C01824=1190.951,366.071,-77.906,-176.070,8.337,148.500
C01825=1190.946,366.351,-77.944,-176.068,8.340,148.500
C01826=1190.942,366.633,-77.983,-176.066,8.344,148.501
C01827=1190.937,366.914,-78.021,-176.065,8.348,148.501
C01828=1190.932,367.161,-78.055,-176.063,8.351,148.502
C01829=1190.929,367.409,-78.090,-176.062,8.354,148.502
C01830=1190.925,367.657,-78.123,-176.060,8.358,148.502
C01831=1190.920,367.904,-78.157,-176.058,8.361,148.503
C01832=1190.917,368.152,-78.191,-176.057,8.364,148.503
C01833=1190.913,368.400,-78.226,-176.055,8.368,148.504
C01834=1190.909,368.647,-78.260,-176.053,8.371,148.504
C01835=1190.904,368.895,-78.294,-176.052,8.374,148.504
C01836=1190.901,369.143,-78.328,-176.050,8.378,148.505
C01837=1190.896,369.390,-78.362,-176.049,8.381,148.505
C01838=1190.893,369.638,-78.396,-176.047,8.385,148.506
C01839=1190.888,369.885,-78.431,-176.046,8.387,148.506
C01840=1190.885,370.134,-78.464,-176.044,8.391,148.507
C01841=1190.880,370.381,-78.499,-176.043,8.394,148.507
C01842=1190.876,370.628,-78.533,-176.041,8.397,148.508
C01843=1190.872,370.876,-78.568,-176.040,8.401,148.508
C01844=1190.869,371.123,-78.602,-176.038,8.404,148.508
C01845=1190.864,371.371,-78.636,-176.037,8.408,148.509
C01846=1190.861,371.619,-78.670,-176.036,8.411,148.509
C01847=1190.856,371.866,-78.705,-176.034,8.414,148.510
C01848=1190.852,372.114,-78.740,-176.033,8.417,148.510
C01849=1190.848,372.362,-78.773,-176.031,8.421,148.511
C01850=1190.843,372.609,-78.807,-176.030,8.424,148.511
C01851=1190.840,372.857,-78.841,-176.029,8.427,148.512
C01852=1190.836,373.105,-78.876,-176.027,8.430,148.512
C01853=1190.832,373.352,-78.910,-176.026,8.433,148.513
C01854=1190.828,373.600,-78.945,-176.025,8.437,148.513
C01855=1190.823,373.847,-78.979,-176.023,8.440,148.513
C01856=1190.820,374.095,-79.013,-176.022,8.444,148.514
C01857=1190.816,374.342,-79.048,-176.021,8.446,148.514
C01858=1190.812,374.591,-79.083,-176.020,8.450,148.515
C01859=1190.808,374.838,-79.116,-176.018,8.453,148.516
C01860=1190.804,375.086,-79.151,-176.017,8.456,148.516
C01861=1190.800,375.333,-79.185,-176.016,8.460,148.517
C01862=1190.796,375.580,-79.220,-176.014,8.463,148.517
C01863=1190.792,375.828,-79.255,-176.013,8.466,148.518
C01864=1190.788,376.075,-79.289,-176.012,8.469,148.518
C01865=1190.784,376.323,-79.324,-176.011,8.473,148.519
C01866=1190.779,376.570,-79.358,-176.010,8.475,148.519
C01867=1190.776,376.818,-79.393,-176.009,8.478,148.520
C01868=1190.772,377.066,-79.427,-176.007,8.482,148.520
C01869=1190.768,377.314,-79.462,-176.006,8.485,148.521
C01870=1190.764,377.561,-79.496,-176.005,8.488,148.521
C01871=1190.760,377.808,-79.531,-176.004,8.492,148.522
C01872=1190.755,378.056,-79.566,-176.002,8.495,148.522
C01873=1190.752,378.304,-79.601,-176.002,8.498,148.523
C01874=1190.748,378.551,-79.634,-176.001,8.501,148.523
C01875=1190.744,378.799,-79.669,-175.999,8.505,148.524
C01876=1190.739,379.047,-79.704,-175.998,8.508,148.524
C01877=1190.735,379.294,-79.739,-175.997,8.510,148.525
C01878=1190.732,379.541,-79.773,-175.996,8.513,148.525
C01879=1190.728,379.789,-79.808,-175.995,8.517,148.526
C01880=1190.723,380.037,-79.842,-175.995,8.520,148.526
C01881=1190.719,380.284,-79.878,-175.993,8.523,148.527
C01882=1190.716,380.531,-79.912,-175.992,8.526,148.527
C01883=1190.712,380.779,-79.947,-175.991,8.530,148.528
C01884=1190.707,381.027,-79.981,-175.990,8.532,148.528
C01885=1190.703,381.274,-80.017,-175.989,8.535,148.529
C01886=1190.700,381.522,-80.051,-175.988,8.539,148.529
C01887=1190.696,381.770,-80.085,-175.988,8.542,148.530
C01888=1190.691,382.017,-80.120,-175.986,8.544,148.530
C01889=1190.687,382.265,-80.155,-175.986,8.548,148.531
C01890=1190.683,382.512,-80.190,-175.985,8.551,148.532
C01891=1190.680,382.760,-80.224,-175.984,8.554,148.532
C01892=1190.675,383.007,-80.259,-175.983,8.557,148.533
C01893=1190.671,383.255,-80.294,-175.982,8.560,148.533
C01894=1190.667,383.502,-80.329,-175.981,8.563,148.534
C01895=1190.663,383.750,-80.364,-175.980,8.566,148.534
C01896=1190.659,383.998,-80.399,-175.980,8.569,148.535
C01897=1190.656,384.244,-80.434,-175.979,8.572,148.535
C01898=1190.652,384.492,-80.468,-175.978,8.575,148.536
C01899=1190.647,384.740,-80.503,-175.977,8.578,148.537
C01900=1190.643,384.987,-80.538,-175.976,8.581,148.537
C01901=1190.639,385.235,-80.573,-175.976,8.584,148.538
C01902=1190.635,385.482,-80.608,-175.975,8.587,148.538
C01903=1190.631,385.730,-80.643,-175.974,8.591,148.539
C01904=1190.627,385.978,-80.678,-175.974,8.593,148.540
C01905=1190.624,386.225,-80.713,-175.973,8.596,148.540
C01906=1190.619,386.472,-80.747,-175.972,8.599,148.541
C01907=1190.615,386.720,-80.783,-175.971,8.602,148.541
C01908=1190.611,386.967,-80.817,-175.970,8.605,148.542
C01909=1190.607,387.215,-80.853,-175.970,8.608,148.542
C01910=1190.603,387.463,-80.888,-175.969,8.611,148.543
C01911=1190.599,387.710,-80.923,-175.969,8.614,148.544
C01912=1190.595,387.958,-80.958,-175.968,8.617,148.544
C01913=1190.591,388.205,-80.993,-175.968,8.619,148.545
C01914=1190.587,388.453,-81.028,-175.967,8.622,148.545
C01915=1190.584,388.700,-81.063,-175.966,8.625,148.546
C01916=1190.579,388.947,-81.097,-175.966,8.628,148.546
C01917=1190.576,389.195,-81.133,-175.965,8.631,148.547
C01918=1190.571,389.442,-81.167,-175.964,8.634,148.548
C01919=1190.567,389.690,-81.203,-175.964,8.636,148.548
C01920=1190.563,389.938,-81.237,-175.963,8.639,148.549
C01921=1190.559,390.185,-81.273,-175.962,8.642,148.549
C01922=1190.555,390.433,-81.307,-175.963,8.645,148.550
C01923=1190.552,390.680,-81.343,-175.962,8.648,148.551
C01924=1190.547,390.927,-81.378,-175.961,8.650,148.551
C01925=1190.543,391.175,-81.413,-175.961,8.653,148.552
C01926=1190.540,391.423,-81.449,-175.960,8.655,148.552
C01927=1190.535,391.670,-81.483,-175.960,8.659,148.553
C01928=1190.531,391.954,-81.524,-175.959,8.662,148.554
C01929=1190.527,392.237,-81.563,-175.958,8.665,148.554
C01930=1190.522,392.520,-81.604,-175.959,8.668,148.555
C01931=1190.517,392.804,-81.644,-175.958,8.671,148.555
C01932=1190.513,393.051,-81.679,-175.957,8.674,148.556
C01933=1190.510,393.299,-81.715,-175.957,8.676,148.557
C01934=1190.505,393.546,-81.749,-175.956,8.680,148.557
C01935=1190.501,393.794,-81.785,-175.956,8.682,148.558
C01936=1190.498,394.041,-81.820,-175.956,8.684,148.558
C01937=1190.493,394.289,-81.855,-175.955,8.687,148.559
C01938=1190.489,394.536,-81.890,-175.955,8.689,148.560
C01939=1190.486,394.784,-81.926,-175.954,8.693,148.560
C01940=1190.481,395.031,-81.960,-175.954,8.695,148.561
C01941=1190.478,395.279,-81.996,-175.954,8.697,148.561
C01942=1190.474,395.526,-82.031,-175.953,8.700,148.562
C01943=1190.469,395.774,-82.066,-175.953,8.703,148.562
C01944=1190.466,396.021,-82.102,-175.953,8.705,148.563
C01945=1190.462,396.269,-82.137,-175.952,8.708,148.564
C01946=1190.457,396.516,-82.173,-175.952,8.711,148.564
C01947=1190.453,396.764,-82.208,-175.952,8.713,148.565
C01948=1190.449,397.011,-82.243,-175.952,8.715,148.565
C01949=1190.445,397.258,-82.278,-175.951,8.718,148.566
C01950=1190.441,397.506,-82.313,-175.951,8.721,148.567
C01951=1190.438,397.754,-82.349,-175.951,8.723,148.567
C01952=1190.433,398.000,-82.384,-175.951,8.725,148.568
C01953=1190.430,398.248,-82.420,-175.950,8.728,148.568
C01954=1190.426,398.496,-82.454,-175.950,8.731,148.569
C01955=1190.421,398.743,-82.490,-175.950,8.733,148.570
C01956=1190.418,398.990,-82.525,-175.949,8.736,148.570
C01957=1190.414,399.238,-82.561,-175.949,8.738,148.571
C01958=1190.410,399.485,-82.596,-175.949,8.740,148.571
C01959=1190.405,399.733,-82.631,-175.949,8.744,148.572
C01960=1190.401,399.981,-82.667,-175.948,8.746,148.572
C01961=1190.398,400.228,-82.702,-175.948,8.748,148.573
C01962=1190.393,400.475,-82.737,-175.948,8.750,148.574
C01963=1190.390,400.722,-82.773,-175.948,8.753,148.574
C01964=1190.386,400.971,-82.808,-175.948,8.755,148.575
C01965=1190.382,401.218,-82.843,-175.948,8.757,148.575
C01966=1190.378,401.465,-82.879,-175.947,8.760,148.576
C01967=1190.374,401.712,-82.914,-175.947,8.763,148.576
C01968=1190.370,401.960,-82.950,-175.946,8.765,148.577
C01969=1190.365,402.208,-82.985,-175.947,8.768,148.578
C01970=1190.362,402.455,-83.020,-175.946,8.770,148.578
C01971=1190.358,402.703,-83.056,-175.946,8.772,148.579
C01972=1190.354,402.950,-83.091,-175.946,8.774,148.579
C01973=1190.350,403.197,-83.127,-175.946,8.777,148.580
C01974=1190.346,403.444,-83.162,-175.946,8.779,148.581
C01975=1190.342,403.692,-83.198,-175.945,8.781,148.581
C01976=1190.338,403.940,-83.233,-175.945,8.784,148.582
C01977=1190.334,404.187,-83.268,-175.945,8.786,148.582
C01978=1190.330,404.435,-83.304,-175.945,8.788,148.583
C01979=1190.326,404.682,-83.339,-175.944,8.791,148.583
C01980=1190.323,404.930,-83.375,-175.945,8.793,148.584
C01981=1190.318,405.177,-83.411,-175.944,8.795,148.584
C01982=1190.314,405.424,-83.446,-175.944,8.798,148.585
C01983=1190.310,405.672,-83.482,-175.944,8.800,148.585
C01984=1190.307,405.919,-83.517,-175.944,8.802,148.586
C01985=1190.302,406.166,-83.553,-175.944,8.804,148.586
C01986=1190.299,406.414,-83.587,-175.944,8.806,148.587
C01987=1190.294,406.662,-83.624,-175.944,8.808,148.588
C01988=1190.290,406.909,-83.659,-175.944,8.811,148.588
C01989=1190.286,407.156,-83.694,-175.943,8.813,148.589
C01990=1190.283,407.404,-83.730,-175.943,8.815,148.589
C01991=1190.279,407.651,-83.765,-175.943,8.818,148.590
C01992=1190.274,407.899,-83.801,-175.943,8.820,148.590
C01993=1190.270,408.146,-83.837,-175.943,8.822,148.591
C01994=1190.267,408.393,-83.872,-175.943,8.824,148.591
C01995=1190.263,408.641,-83.908,-175.943,8.826,148.592
C01996=1190.259,408.888,-83.943,-175.943,8.828,148.593
C01997=1190.254,409.135,-83.979,-175.942,8.831,148.593
C01998=1190.251,409.383,-84.015,-175.942,8.833,148.594
C01999=1190.247,409.630,-84.050,-175.942,8.835,148.594
C02000=1190.243,409.878,-84.086,-175.942,8.837,148.595
C02001=1190.240,410.125,-84.121,-175.942,8.839,148.595
C02002=1190.235,410.373,-84.157,-175.942,8.841,148.596
C02003=1190.231,410.620,-84.193,-175.942,8.844,148.596
C02004=1190.227,410.868,-84.228,-175.942,8.846,148.597
C02005=1190.224,411.115,-84.264,-175.941,8.848,148.597
C02006=1190.220,411.363,-84.299,-175.942,8.850,148.598
C02007=1190.215,411.610,-84.335,-175.941,8.852,148.598
C02008=1190.211,411.857,-84.371,-175.941,8.854,148.599
C02009=1190.208,412.105,-84.406,-175.941,8.856,148.599
C02010=1190.204,412.352,-84.442,-175.941,8.858,148.600
C02011=1190.199,412.599,-84.477,-175.941,8.860,148.600
C02012=1190.195,412.847,-84.513,-175.941,8.862,148.601
C02013=1190.192,413.094,-84.549,-175.941,8.865,148.601
C02014=1190.188,413.342,-84.584,-175.941,8.866,148.602
C02015=1190.184,413.590,-84.620,-175.941,8.868,148.602
C02016=1190.179,413.836,-84.655,-175.940,8.871,148.603
C02017=1190.176,414.084,-84.691,-175.940,8.873,148.603
C02018=1190.171,414.332,-84.727,-175.941,8.875,148.604
C02019=1190.168,414.579,-84.763,-175.941,8.877,148.605
C02020=1190.164,414.827,-84.798,-175.940,8.879,148.605
C02021=1190.160,415.074,-84.833,-175.941,8.881,148.606
C02022=1190.155,415.321,-84.870,-175.940,8.883,148.606
C02023=1190.152,415.569,-84.905,-175.940,8.885,148.607
C02024=1190.146,415.957,-84.961,-175.940,8.888,148.607
C02025=1190.142,416.344,-85.018,-175.940,8.891,148.608
C02026=1190.142,416.732,-85.072,-175.939,8.894,148.609
C02027=1190.144,417.119,-85.127,-175.939,8.897,148.610
C02028=1189.723,417.119,-85.168,-175.942,8.907,148.613
C02029=1189.720,416.730,-85.112,-175.943,8.905,148.613
C02030=1189.721,416.339,-85.057,-175.943,8.902,148.612
C02031=1189.724,415.948,-85.001,-175.943,8.898,148.611
C02032=1189.731,415.557,-84.945,-175.943,8.896,148.610
C02033=1189.734,415.310,-84.909,-175.943,8.893,148.610
C02034=1189.738,415.063,-84.872,-175.944,8.891,148.609
C02035=1189.743,414.816,-84.837,-175.943,8.890,148.609
C02036=1189.746,414.568,-84.801,-175.944,8.888,148.608
C02037=1189.750,414.321,-84.766,-175.944,8.885,148.608
C02038=1189.754,414.073,-84.730,-175.944,8.884,148.607
C02039=1189.758,413.825,-84.694,-175.944,8.882,148.607
C02040=1189.762,413.579,-84.659,-175.944,8.879,148.606
C02041=1189.766,413.331,-84.623,-175.944,8.877,148.606
C02042=1189.770,413.083,-84.587,-175.944,8.875,148.605
C02043=1189.774,412.836,-84.552,-175.944,8.873,148.605
C02044=1189.778,412.588,-84.516,-175.944,8.871,148.604
C02045=1189.782,412.342,-84.481,-175.944,8.869,148.604
C02046=1189.786,412.094,-84.445,-175.944,8.867,148.603
C02047=1189.790,411.846,-84.409,-175.944,8.865,148.603
C02048=1189.794,411.599,-84.374,-175.945,8.863,148.602
C02049=1189.797,411.351,-84.338,-175.945,8.860,148.602
C02050=1189.802,411.104,-84.302,-175.945,8.859,148.601
C02051=1189.806,410.857,-84.267,-175.945,8.857,148.601
C02052=1189.810,410.609,-84.231,-175.945,8.854,148.600
C02053=1189.813,410.362,-84.196,-175.945,8.852,148.599
C02054=1189.818,410.114,-84.160,-175.945,8.850,148.599
C02055=1189.822,409.867,-84.124,-175.945,8.848,148.598
C02056=1189.826,409.620,-84.089,-175.945,8.846,148.598
C02057=1189.829,409.372,-84.053,-175.945,8.844,148.597
C02058=1189.833,409.125,-84.018,-175.946,8.841,148.597
C02059=1189.838,408.877,-83.982,-175.946,8.839,148.596
C02060=1189.842,408.630,-83.947,-175.945,8.838,148.596
C02061=1189.845,408.382,-83.911,-175.946,8.835,148.595
C02062=1189.849,408.135,-83.875,-175.946,8.833,148.594
C02063=1189.853,407.887,-83.839,-175.946,8.830,148.594
C02064=1189.858,407.640,-83.804,-175.946,8.828,148.593
C02065=1189.861,407.393,-83.769,-175.946,8.826,148.593
C02066=1189.865,407.145,-83.733,-175.947,8.824,148.592
C02067=1189.869,406.898,-83.697,-175.946,8.822,148.592
C02068=1189.873,406.651,-83.662,-175.946,8.820,148.591
C02069=1189.877,406.403,-83.626,-175.946,8.817,148.591
C02070=1189.881,406.156,-83.591,-175.947,8.815,148.590
C02071=1189.885,405.908,-83.555,-175.947,8.813,148.590
C02072=1189.889,405.661,-83.520,-175.947,8.811,148.589
C02073=1189.892,405.414,-83.484,-175.947,8.808,148.589
C02074=1189.897,405.165,-83.449,-175.948,8.806,148.588
C02075=1189.901,404.918,-83.413,-175.947,8.803,148.587
C02076=1189.905,404.671,-83.378,-175.948,8.801,148.587
C02077=1189.909,404.424,-83.343,-175.948,8.799,148.586
C02078=1189.912,404.176,-83.307,-175.948,8.797,148.586
C02079=1189.916,403.929,-83.271,-175.948,8.794,148.585
C02080=1189.921,403.682,-83.236,-175.948,8.792,148.584
C02081=1189.925,403.434,-83.200,-175.948,8.790,148.584
C02082=1189.928,403.187,-83.165,-175.949,8.787,148.583
C02083=1189.932,402.938,-83.130,-175.949,8.785,148.583
C02084=1189.937,402.692,-83.095,-175.949,8.783,148.582
C02085=1189.940,402.444,-83.059,-175.949,8.780,148.582
C02086=1189.944,402.197,-83.024,-175.949,8.778,148.581
C02087=1189.948,401.949,-82.987,-175.949,8.776,148.581
C02088=1189.953,401.702,-82.952,-175.950,8.773,148.580
C02089=1189.956,401.455,-82.917,-175.950,8.771,148.580
C02090=1189.960,401.206,-82.882,-175.950,8.769,148.579
C02091=1189.965,400.960,-82.847,-175.950,8.766,148.578
C02092=1189.968,400.712,-82.811,-175.950,8.764,148.578
C02093=1189.972,400.465,-82.776,-175.950,8.762,148.577
C02094=1189.976,400.217,-82.740,-175.951,8.758,148.576
C02095=1189.981,399.969,-82.705,-175.951,8.756,148.576
C02096=1189.985,399.722,-82.669,-175.951,8.754,148.575
C02097=1189.988,399.474,-82.634,-175.952,8.752,148.575
C02098=1189.992,399.228,-82.599,-175.952,8.749,148.574
C02099=1189.996,398.980,-82.563,-175.952,8.747,148.574
C02100=1190.000,398.732,-82.528,-175.952,8.744,148.573
C02101=1190.004,398.484,-82.493,-175.953,8.741,148.573
C02102=1190.008,398.238,-82.458,-175.953,8.739,148.572
C02103=1190.012,397.990,-82.422,-175.953,8.737,148.571
C02104=1190.016,397.742,-82.387,-175.953,8.734,148.571
C02105=1190.021,397.495,-82.351,-175.954,8.731,148.570
C02106=1190.024,397.247,-82.316,-175.954,8.729,148.570
C02107=1190.028,397.000,-82.280,-175.954,8.727,148.569
C02108=1190.033,396.752,-82.246,-175.954,8.724,148.568
C02109=1190.036,396.505,-82.210,-175.955,8.721,148.568
C02110=1190.040,396.257,-82.175,-175.955,8.719,148.567
C02111=1190.044,396.011,-82.140,-175.955,8.716,148.567
C02112=1190.048,395.763,-82.105,-175.956,8.713,148.566
C02113=1190.052,395.515,-82.069,-175.956,8.711,148.565
C02114=1190.056,395.268,-82.034,-175.956,8.709,148.565
C02115=1190.060,395.020,-81.999,-175.957,8.705,148.564
C02116=1190.064,394.773,-81.964,-175.957,8.703,148.564
C02117=1190.068,394.526,-81.928,-175.957,8.701,148.563
C02118=1190.072,394.278,-81.893,-175.958,8.698,148.562
C02119=1190.076,394.030,-81.858,-175.958,8.695,148.562
C02120=1190.080,393.783,-81.823,-175.958,8.693,148.561
C02121=1190.083,393.536,-81.787,-175.959,8.690,148.561
C02122=1190.087,393.288,-81.752,-175.959,8.687,148.560
C02123=1190.092,393.041,-81.717,-175.960,8.684,148.560
C02124=1190.096,392.793,-81.682,-175.960,8.682,148.559
C02125=1190.100,392.510,-81.642,-175.961,8.679,148.558
C02126=1190.105,392.226,-81.601,-175.961,8.675,148.558
C02127=1190.109,391.942,-81.561,-175.962,8.672,148.557
C02128=1190.114,391.659,-81.520,-175.962,8.669,148.556
C02129=1190.118,391.411,-81.486,-175.963,8.667,148.556
C02130=1190.122,391.164,-81.450,-175.963,8.664,148.555
C02131=1190.126,390.916,-81.416,-175.964,8.661,148.555
C02132=1190.130,390.669,-81.380,-175.964,8.658,148.554
C02133=1190.134,390.421,-81.344,-175.964,8.656,148.553
C02134=1190.138,390.174,-81.311,-175.965,8.653,148.553
C02135=1190.141,389.927,-81.275,-175.966,8.649,148.552
C02136=1190.146,389.679,-81.241,-175.966,8.647,148.552
C02137=1190.150,389.432,-81.205,-175.967,8.644,148.551
C02138=1190.153,389.184,-81.170,-175.967,8.642,148.551
C02139=1190.158,388.937,-81.135,-175.968,8.639,148.550
C02140=1190.162,388.689,-81.100,-175.969,8.636,148.549
C02141=1190.165,388.441,-81.065,-175.969,8.633,148.549
C02142=1190.170,388.194,-81.030,-175.969,8.630,148.548
C02143=1190.174,387.946,-80.995,-175.970,8.627,148.547
C02144=1190.178,387.699,-80.960,-175.971,8.624,148.547
C02145=1190.182,387.452,-80.925,-175.971,8.622,148.546
C02146=1190.186,387.203,-80.890,-175.972,8.618,148.546
C02147=1190.190,386.957,-80.855,-175.973,8.615,148.545
C02148=1190.194,386.708,-80.820,-175.974,8.612,148.545
C02149=1190.198,386.462,-80.785,-175.974,8.610,148.544
C02150=1190.202,386.214,-80.750,-175.975,8.607,148.543
C02151=1190.205,385.966,-80.715,-175.975,8.604,148.543
C02152=1190.210,385.719,-80.680,-175.976,8.601,148.542
C02153=1190.213,385.471,-80.645,-175.977,8.598,148.542
C02154=1190.218,385.224,-80.610,-175.978,8.594,148.541
C02155=1190.222,384.977,-80.575,-175.978,8.592,148.541
C02156=1190.226,384.729,-80.540,-175.979,8.589,148.540
C02157=1190.229,384.481,-80.506,-175.980,8.586,148.540
C02158=1190.233,384.234,-80.471,-175.981,8.583,148.539
C02159=1190.238,383.986,-80.436,-175.982,8.580,148.538
C02160=1190.241,383.739,-80.401,-175.983,8.577,148.538
C02161=1190.246,383.491,-80.366,-175.983,8.574,148.537
C02162=1190.250,383.243,-80.331,-175.984,8.571,148.537
C02163=1190.253,382.997,-80.297,-175.985,8.568,148.536
C02164=1190.257,382.749,-80.262,-175.986,8.565,148.536
C02165=1190.262,382.501,-80.227,-175.987,8.562,148.535
C02166=1190.266,382.254,-80.192,-175.988,8.559,148.535
C02167=1190.270,382.006,-80.157,-175.989,8.556,148.534
C02168=1190.274,381.758,-80.122,-175.989,8.553,148.533
C02169=1190.277,381.511,-80.088,-175.990,8.549,148.533
C02170=1190.282,381.264,-80.053,-175.991,8.547,148.532
C02171=1190.286,381.016,-80.018,-175.993,8.543,148.532
C02172=1190.290,380.768,-79.984,-175.994,8.540,148.531
C02173=1190.294,380.521,-79.948,-175.994,8.536,148.531
C02174=1190.298,380.274,-79.914,-175.996,8.534,148.530
C02175=1190.302,380.025,-79.880,-175.996,8.531,148.530
C02176=1190.306,379.779,-79.844,-175.997,8.528,148.529
C02177=1190.310,379.530,-79.809,-175.998,8.525,148.529
C02178=1190.314,379.283,-79.776,-176.000,8.521,148.528
C02179=1190.318,379.035,-79.741,-176.001,8.518,148.527
C02180=1190.322,378.788,-79.706,-176.002,8.515,148.527
C02181=1190.326,378.540,-79.671,-176.003,8.512,148.526
C02182=1190.330,378.293,-79.637,-176.003,8.509,148.526
C02183=1190.334,378.045,-79.602,-176.005,8.505,148.525
C02184=1190.338,377.798,-79.568,-176.006,8.502,148.525
C02185=1190.342,377.550,-79.533,-176.007,8.499,148.524
C02186=1190.346,377.302,-79.499,-176.008,8.496,148.524
C02187=1190.350,377.055,-79.463,-176.009,8.492,148.523
C02188=1190.354,376.808,-79.429,-176.011,8.489,148.523
C02189=1190.358,376.560,-79.395,-176.011,8.486,148.522
C02190=1190.362,376.312,-79.360,-176.013,8.483,148.522
C02191=1190.367,376.065,-79.326,-176.014,8.480,148.521
C02192=1190.370,375.817,-79.291,-176.015,8.477,148.521
C02193=1190.374,375.570,-79.257,-176.017,8.473,148.520
C02194=1190.378,375.322,-79.222,-176.018,8.470,148.520
C02195=1190.382,375.074,-79.188,-176.019,8.467,148.519
C02196=1190.386,374.826,-79.153,-176.020,8.463,148.519
C02197=1190.391,374.579,-79.118,-176.022,8.460,148.518
C02198=1190.394,374.332,-79.084,-176.023,8.457,148.518
C02199=1190.398,374.084,-79.050,-176.024,8.454,148.517
C02200=1190.402,373.837,-79.016,-176.026,8.451,148.517
C02201=1190.406,373.589,-78.981,-176.027,8.447,148.516
C02202=1190.411,373.342,-78.946,-176.028,8.444,148.516
C02203=1190.414,373.094,-78.912,-176.030,8.441,148.516
C02204=1190.418,372.846,-78.878,-176.031,8.437,148.515
C02205=1190.422,372.599,-78.843,-176.033,8.434,148.515
C02206=1190.426,372.351,-78.809,-176.034,8.431,148.514
C02207=1190.431,372.103,-78.775,-176.036,8.427,148.514
C02208=1190.434,371.855,-78.741,-176.036,8.424,148.513
C02209=1190.439,371.608,-78.707,-176.038,8.421,148.513
C02210=1190.442,371.360,-78.672,-176.039,8.418,148.512
C02211=1190.447,371.113,-78.638,-176.041,8.414,148.512
C02212=1190.451,370.866,-78.604,-176.042,8.411,148.511
C02213=1190.455,370.617,-78.569,-176.044,8.408,148.511
C02214=1190.458,370.370,-78.535,-176.045,8.405,148.510
C02215=1190.463,370.123,-78.501,-176.047,8.401,148.510
C02216=1190.466,369.875,-78.467,-176.048,8.398,148.510
C02217=1190.471,369.627,-78.433,-176.050,8.395,148.509
C02218=1190.474,369.379,-78.399,-176.052,8.391,148.509
C02219=1190.479,369.132,-78.364,-176.052,8.388,148.508
C02220=1190.483,368.885,-78.330,-176.054,8.384,148.508
C02221=1190.487,368.637,-78.295,-176.055,8.382,148.507
C02222=1190.491,368.389,-78.262,-176.057,8.378,148.507
C02223=1190.495,368.141,-78.228,-176.059,8.374,148.506
C02224=1190.499,367.894,-78.194,-176.060,8.371,148.506
C02225=1190.503,367.646,-78.159,-176.062,8.368,148.506
C02226=1190.507,367.398,-78.126,-176.063,8.365,148.505
C02227=1190.511,367.150,-78.091,-176.065,8.361,148.505
C02228=1190.515,366.903,-78.057,-176.067,8.358,148.504
C02229=1190.520,366.623,-78.019,-176.069,8.354,148.504
C02230=1190.524,366.341,-77.980,-176.071,8.351,148.504
C02231=1190.530,366.060,-77.942,-176.072,8.347,148.503
C02232=1190.534,365.778,-77.903,-176.074,8.343,148.503
C02233=1190.538,365.531,-77.869,-176.076,8.340,148.502
C02234=1190.541,365.283,-77.835,-176.078,8.336,148.502
C02235=1190.546,365.035,-77.801,-176.079,8.333,148.501
C02236=1190.550,364.788,-77.767,-176.081,8.330,148.501
C02237=1190.554,364.541,-77.734,-176.083,8.326,148.501
C02238=1190.558,364.293,-77.699,-176.085,8.323,148.500
C02239=1190.562,364.045,-77.665,-176.086,8.320,148.500
C02240=1190.567,363.797,-77.631,-176.088,8.316,148.499
C02241=1190.570,363.550,-77.597,-176.090,8.313,148.499
C02242=1190.574,363.302,-77.564,-176.092,8.309,148.499
C02243=1190.578,363.055,-77.530,-176.093,8.306,148.498
C02244=1190.583,362.807,-77.496,-176.095,8.303,148.498
C02245=1190.586,362.559,-77.462,-176.097,8.299,148.498
C02246=1190.590,362.311,-77.429,-176.099,8.296,148.497
C02247=1190.595,362.064,-77.394,-176.100,8.293,148.497
C02248=1190.599,361.816,-77.361,-176.102,8.289,148.497
C02249=1190.602,361.568,-77.327,-176.104,8.286,148.496
C02250=1190.606,361.320,-77.294,-176.106,8.282,148.496
C02251=1190.611,361.073,-77.259,-176.107,8.280,148.495
C02252=1190.615,360.825,-77.226,-176.109,8.276,148.495
C02253=1190.619,360.578,-77.192,-176.111,8.273,148.495
C02254=1190.622,360.330,-77.159,-176.114,8.269,148.495
C02255=1190.627,360.082,-77.125,-176.115,8.266,148.494
C02256=1190.631,359.835,-77.091,-176.117,8.263,148.494
C02257=1190.635,359.587,-77.058,-176.119,8.260,148.494
C02258=1190.639,359.340,-77.024,-176.121,8.256,148.493
C02259=1190.643,359.091,-76.990,-176.123,8.253,148.493
C02260=1190.647,358.843,-76.957,-176.125,8.249,148.492
C02261=1190.651,358.596,-76.923,-176.127,8.246,148.492
C02262=1190.655,358.348,-76.890,-176.128,8.243,148.492
C02263=1190.659,358.101,-76.857,-176.130,8.240,148.492
C02264=1190.663,357.854,-76.823,-176.132,8.236,148.491
C02265=1190.667,357.605,-76.789,-176.134,8.233,148.491
C02266=1190.672,357.357,-76.756,-176.136,8.229,148.491
C02267=1190.676,357.109,-76.722,-176.138,8.226,148.490
C02268=1190.680,356.862,-76.689,-176.141,8.222,148.490
C02269=1190.684,356.615,-76.655,-176.142,8.219,148.490
C02270=1190.688,356.367,-76.622,-176.144,8.216,148.489
C02271=1190.692,356.119,-76.589,-176.146,8.213,148.489
C02272=1190.696,355.871,-76.554,-176.148,8.209,148.489
C02273=1190.700,355.623,-76.521,-176.150,8.206,148.489
C02274=1190.704,355.376,-76.488,-176.152,8.202,148.488
C02275=1190.708,355.128,-76.455,-176.154,8.199,148.488
C02276=1190.712,354.880,-76.422,-176.157,8.196,148.488
C02277=1190.717,354.632,-76.389,-176.158,8.193,148.487
C02278=1190.720,354.385,-76.355,-176.160,8.190,148.487
C02279=1190.725,354.138,-76.321,-176.162,8.186,148.487
C02280=1190.729,353.890,-76.288,-176.164,8.183,148.486
C02281=1190.732,353.641,-76.255,-176.166,8.179,148.486
C02282=1190.736,353.394,-76.222,-176.169,8.176,148.486
C02283=1190.741,353.146,-76.189,-176.171,8.173,148.486
C02284=1190.745,352.898,-76.155,-176.172,8.170,148.485
C02285=1190.749,352.650,-76.122,-176.174,8.167,148.485
C02286=1190.753,352.403,-76.089,-176.177,8.163,148.485
C02287=1190.757,352.155,-76.056,-176.179,8.160,148.485
C02288=1190.761,351.907,-76.023,-176.181,8.156,148.484
C02289=1190.765,351.660,-75.990,-176.183,8.153,148.484
C02290=1190.769,351.412,-75.956,-176.185,8.150,148.484
C02291=1190.774,351.164,-75.923,-176.187,8.146,148.484
C02292=1190.778,350.916,-75.890,-176.189,8.144,148.483
C02293=1190.782,350.669,-75.857,-176.191,8.140,148.483
C02294=1190.786,350.421,-75.824,-176.193,8.137,148.483
C02295=1190.790,350.173,-75.791,-176.195,8.133,148.483
C02296=1190.794,349.925,-75.757,-176.198,8.130,148.482
C02297=1190.798,349.678,-75.724,-176.200,8.127,148.482
C02298=1190.803,349.429,-75.692,-176.202,8.123,148.482
C02299=1190.807,349.182,-75.659,-176.204,8.121,148.482
C02300=1190.811,348.934,-75.626,-176.206,8.117,148.481
C02301=1190.815,348.686,-75.593,-176.208,8.114,148.481
C02302=1190.819,348.439,-75.560,-176.210,8.111,148.481
C02303=1190.823,348.191,-75.527,-176.212,8.107,148.481
C02304=1190.827,347.943,-75.494,-176.215,8.104,148.480
C02305=1190.831,347.695,-75.461,-176.217,8.101,148.480
C02306=1190.836,347.447,-75.428,-176.219,8.098,148.480
C02307=1190.840,347.199,-75.395,-176.221,8.095,148.480
C02308=1190.843,346.952,-75.362,-176.223,8.092,148.480
C02309=1190.848,346.704,-75.330,-176.225,8.088,148.479
C02310=1190.852,346.456,-75.297,-176.228,8.085,148.479
C02311=1190.856,346.208,-75.263,-176.230,8.082,148.479
C02312=1190.860,345.960,-75.231,-176.232,8.078,148.479
C02313=1190.864,345.712,-75.198,-176.234,8.075,148.478
C02314=1190.868,345.465,-75.165,-176.236,8.072,148.478
C02315=1190.873,345.218,-75.133,-176.238,8.069,148.478
C02316=1190.877,344.969,-75.100,-176.240,8.066,148.478
C02317=1190.881,344.722,-75.067,-176.243,8.063,148.478
C02318=1190.885,344.474,-75.035,-176.245,8.059,148.477
C02319=1190.889,344.226,-75.002,-176.247,8.056,148.477
C02320=1190.893,343.978,-74.969,-176.249,8.053,148.477
C02321=1190.898,343.730,-74.936,-176.251,8.050,148.477
C02322=1190.901,343.482,-74.904,-176.253,8.047,148.477
C02323=1190.905,343.234,-74.871,-176.256,8.043,148.476
C02324=1190.910,342.986,-74.838,-176.258,8.040,148.476
C02325=1190.915,342.739,-74.806,-176.260,8.037,148.476
C02326=1190.918,342.491,-74.774,-176.262,8.033,148.476
C02327=1190.922,342.244,-74.740,-176.265,8.030,148.475
C02328=1190.927,341.995,-74.708,-176.267,8.028,148.476
C02329=1190.930,341.748,-74.675,-176.269,8.025,148.475
C02330=1190.934,341.499,-74.643,-176.271,8.021,148.475
C02331=1190.939,341.252,-74.611,-176.273,8.018,148.475
C02332=1190.943,341.004,-74.578,-176.276,8.015,148.475
C02333=1190.947,340.726,-74.542,-176.278,8.011,148.474
C02334=1190.953,340.447,-74.505,-176.281,8.007,148.474
C02335=1190.957,340.168,-74.469,-176.283,8.004,148.474
C02336=1190.962,339.889,-74.432,-176.286,8.001,148.474
C02337=1190.965,339.642,-74.400,-176.288,7.997,148.474
C02338=1190.970,339.393,-74.367,-176.290,7.994,148.474
C02339=1190.974,339.145,-74.335,-176.292,7.991,148.473
C02340=1190.978,338.898,-74.303,-176.295,7.987,148.473
C02341=1190.982,338.650,-74.270,-176.297,7.985,148.473
C02342=1190.986,338.402,-74.238,-176.299,7.982,148.473
C02343=1190.990,338.154,-74.205,-176.301,7.979,148.473
C02344=1190.995,337.907,-74.174,-176.303,7.975,148.472
C02345=1190.999,337.659,-74.141,-176.306,7.972,148.472
C02346=1191.003,337.410,-74.109,-176.308,7.969,148.472
C02347=1191.007,337.163,-74.076,-176.311,7.966,148.472
C02348=1191.011,336.914,-74.044,-176.312,7.963,148.472
C02349=1191.016,336.667,-74.012,-176.315,7.960,148.472
C02350=1191.020,336.419,-73.980,-176.317,7.957,148.472
C02351=1191.024,336.171,-73.947,-176.320,7.953,148.471
C02352=1191.027,335.923,-73.915,-176.322,7.950,148.471
C02353=1191.032,335.676,-73.883,-176.324,7.947,148.471
C02354=1191.036,335.428,-73.851,-176.327,7.944,148.471
C02355=1191.040,335.179,-73.819,-176.328,7.941,148.471
C02356=1191.044,334.931,-73.787,-176.331,7.938,148.471
C02357=1191.049,334.684,-73.754,-176.333,7.935,148.471
C02358=1191.053,334.436,-73.723,-176.336,7.932,148.470
C02359=1191.057,334.188,-73.690,-176.338,7.928,148.470
C02360=1191.061,333.940,-73.659,-176.340,7.925,148.470
C02361=1191.065,333.692,-73.627,-176.342,7.923,148.470
C02362=1191.069,333.444,-73.594,-176.344,7.919,148.470
C02363=1191.073,333.196,-73.563,-176.347,7.916,148.470
C02364=1191.078,332.948,-73.530,-176.349,7.913,148.470
C02365=1191.082,332.700,-73.499,-176.352,7.910,148.469
C02366=1191.086,332.452,-73.467,-176.354,7.907,148.469
C02367=1191.091,332.205,-73.435,-176.357,7.903,148.469
C02368=1191.094,331.957,-73.403,-176.359,7.901,148.469
C02369=1191.098,331.709,-73.371,-176.361,7.898,148.469
C02370=1191.103,331.461,-73.339,-176.363,7.895,148.469
C02371=1191.107,331.213,-73.307,-176.366,7.892,148.469
C02372=1191.111,330.965,-73.275,-176.368,7.888,148.469
C02373=1191.116,330.717,-73.243,-176.371,7.885,148.469
C02374=1191.119,330.469,-73.211,-176.372,7.883,148.468
C02375=1191.124,330.222,-73.180,-176.375,7.879,148.468
C02376=1191.128,329.973,-73.147,-176.377,7.876,148.468
C02377=1191.132,329.725,-73.116,-176.380,7.873,148.468
C02378=1191.136,329.478,-73.084,-176.382,7.870,148.468
C02379=1191.140,329.229,-73.053,-176.385,7.867,148.468
C02380=1191.145,328.981,-73.020,-176.386,7.864,148.468
C02381=1191.149,328.734,-72.989,-176.389,7.861,148.468
C02382=1191.153,328.486,-72.957,-176.391,7.858,148.467
C02383=1191.157,328.238,-72.926,-176.394,7.855,148.467
C02384=1191.162,327.989,-72.894,-176.396,7.852,148.467
C02385=1191.165,327.741,-72.862,-176.399,7.849,148.467
C02386=1191.170,327.494,-72.831,-176.401,7.846,148.467
C02387=1191.173,327.246,-72.799,-176.403,7.843,148.467
C02388=1191.178,326.998,-72.768,-176.406,7.840,148.467
C02389=1191.182,326.750,-72.736,-176.408,7.837,148.467
C02390=1191.187,326.502,-72.704,-176.410,7.833,148.467
C02391=1191.190,326.254,-72.672,-176.413,7.830,148.467
C02392=1191.194,326.006,-72.641,-176.415,7.828,148.466
C02393=1191.199,325.758,-72.610,-176.418,7.825,148.466
C02394=1191.202,325.510,-72.578,-176.420,7.822,148.466
C02395=1191.207,325.262,-72.547,-176.422,7.819,148.466
C02396=1191.211,325.014,-72.515,-176.425,7.815,148.466
C02397=1191.216,324.767,-72.483,-176.427,7.812,148.466
C02398=1191.220,324.518,-72.452,-176.429,7.810,148.466
C02399=1191.224,324.271,-72.421,-176.432,7.807,148.466
C02400=1191.228,324.022,-72.389,-176.434,7.803,148.466
C02401=1191.232,323.775,-72.358,-176.437,7.800,148.466
C02402=1191.236,323.527,-72.326,-176.439,7.797,148.465
C02403=1191.241,323.279,-72.295,-176.442,7.794,148.465
C02404=1191.244,323.031,-72.263,-176.444,7.792,148.466
C02405=1191.249,322.783,-72.233,-176.446,7.789,148.465
C02406=1191.253,322.535,-72.201,-176.449,7.786,148.465
C02407=1191.257,322.287,-72.170,-176.451,7.782,148.465
C02408=1191.261,322.039,-72.138,-176.454,7.779,148.465
C02409=1191.266,321.791,-72.107,-176.455,7.777,148.465
C02410=1191.269,321.543,-72.076,-176.458,7.774,148.465
C02411=1191.274,321.295,-72.045,-176.461,7.771,148.465
C02412=1191.278,321.047,-72.013,-176.463,7.767,148.465
C02413=1191.282,320.799,-71.982,-176.466,7.764,148.465
C02414=1191.286,320.550,-71.951,-176.468,7.761,148.465
C02415=1191.291,320.303,-71.920,-176.470,7.759,148.465
C02416=1191.295,320.054,-71.888,-176.473,7.756,148.465
C02417=1191.299,319.807,-71.857,-176.475,7.752,148.464
C02418=1191.304,319.559,-71.826,-176.478,7.749,148.464
C02419=1191.308,319.310,-71.795,-176.480,7.746,148.464
C02420=1191.312,319.063,-71.764,-176.482,7.744,148.464
C02421=1191.316,318.814,-71.733,-176.485,7.741,148.464
C02422=1191.321,318.566,-71.702,-176.487,7.738,148.464
C02423=1191.325,318.317,-71.671,-176.490,7.735,148.464
C02424=1191.329,318.070,-71.639,-176.493,7.732,148.464
C02425=1191.333,317.822,-71.609,-176.495,7.728,148.464
C02426=1191.337,317.574,-71.578,-176.497,7.726,148.464
C02427=1191.341,317.326,-71.546,-176.500,7.723,148.464
C02428=1191.346,317.078,-71.516,-176.502,7.720,148.464
C02429=1191.350,316.830,-71.484,-176.505,7.717,148.464
C02430=1191.354,316.582,-71.454,-176.507,7.714,148.464
C02431=1191.358,316.333,-71.423,-176.509,7.711,148.464
C02432=1191.362,316.086,-71.392,-176.512,7.708,148.464
C02433=1191.366,315.838,-71.361,-176.514,7.705,148.464
C02434=1191.370,315.590,-71.330,-176.517,7.702,148.463
C02435=1191.375,315.342,-71.299,-176.519,7.699,148.463
C02436=1191.380,315.094,-71.268,-176.521,7.697,148.463
C02437=1191.384,314.817,-71.234,-176.525,7.693,148.463
C02438=1191.389,314.541,-71.200,-176.527,7.690,148.463
C02439=1191.393,314.264,-71.165,-176.530,7.687,148.463
C02440=1191.398,313.988,-71.131,-176.532,7.684,148.463
C02441=1191.402,313.740,-71.100,-176.535,7.681,148.463
C02442=1191.407,313.492,-71.069,-176.537,7.677,148.463
C02443=1191.411,313.244,-71.038,-176.540,7.674,148.463
C02444=1191.414,312.995,-71.008,-176.542,7.672,148.463
C02445=1191.419,312.748,-70.977,-176.545,7.669,148.463
C02446=1191.424,312.500,-70.946,-176.547,7.666,148.463
C02447=1191.428,312.251,-70.915,-176.550,7.663,148.463
C02448=1191.432,312.003,-70.885,-176.552,7.660,148.463
C02449=1191.436,311.755,-70.854,-176.555,7.657,148.463
C02450=1191.441,311.507,-70.824,-176.557,7.654,148.463
C02451=1191.444,311.259,-70.793,-176.560,7.651,148.463
C02452=1191.449,311.011,-70.762,-176.562,7.648,148.463
C02453=1191.453,310.763,-70.732,-176.565,7.645,148.463
C02454=1191.457,310.515,-70.702,-176.567,7.643,148.463
C02455=1191.461,310.266,-70.671,-176.569,7.640,148.463
C02456=1191.466,310.018,-70.640,-176.572,7.637,148.463
C02457=1191.470,309.771,-70.610,-176.575,7.634,148.463
C02458=1191.475,309.523,-70.579,-176.576,7.631,148.463
C02459=1191.478,309.274,-70.549,-176.579,7.628,148.463
C02460=1191.482,309.026,-70.518,-176.582,7.625,148.463
C02461=1191.487,308.778,-70.488,-176.585,7.622,148.463
C02462=1191.491,308.530,-70.458,-176.587,7.619,148.463
C02463=1191.496,308.282,-70.427,-176.589,7.617,148.462
C02464=1191.499,308.034,-70.396,-176.592,7.614,148.462
C02465=1191.504,307.785,-70.366,-176.594,7.611,148.462
C02466=1191.508,307.538,-70.336,-176.597,7.608,148.462
C02467=1191.513,307.290,-70.305,-176.599,7.605,148.463
C02468=1191.517,307.042,-70.275,-176.602,7.602,148.463
C02469=1191.521,306.793,-70.245,-176.604,7.599,148.462
C02470=1191.525,306.545,-70.214,-176.607,7.596,148.462
C02471=1191.529,306.297,-70.184,-176.609,7.594,148.462
C02472=1191.534,306.048,-70.154,-176.612,7.591,148.462
C02473=1191.538,305.801,-70.124,-176.614,7.588,148.462
C02474=1191.543,305.553,-70.093,-176.617,7.585,148.462
C02475=1191.547,305.305,-70.064,-176.619,7.582,148.462
C02476=1191.551,305.057,-70.033,-176.622,7.579,148.462
C02477=1191.555,304.808,-70.003,-176.624,7.576,148.462
C02478=1191.560,304.560,-69.972,-176.627,7.573,148.462
C02479=1191.564,304.312,-69.942,-176.630,7.570,148.462
C02480=1191.568,304.064,-69.913,-176.632,7.568,148.462
C02481=1191.572,303.816,-69.882,-176.634,7.565,148.462
C02482=1191.576,303.568,-69.852,-176.637,7.562,148.462
C02483=1191.581,303.320,-69.822,-176.639,7.559,148.462
C02484=1191.585,303.071,-69.792,-176.642,7.557,148.462
C02485=1191.590,302.823,-69.761,-176.644,7.554,148.462
C02486=1191.593,302.574,-69.732,-176.647,7.551,148.462
C02487=1191.597,302.327,-69.701,-176.650,7.548,148.462
C02488=1191.602,302.078,-69.671,-176.652,7.545,148.462
C02489=1191.606,301.831,-69.641,-176.654,7.542,148.462
C02490=1191.610,301.582,-69.612,-176.657,7.539,148.462
C02491=1191.615,301.334,-69.582,-176.660,7.536,148.462
C02492=1191.619,301.086,-69.551,-176.662,7.534,148.462
C02493=1191.623,300.838,-69.522,-176.664,7.531,148.462
C02494=1191.628,300.590,-69.491,-176.667,7.528,148.462
C02495=1191.632,300.342,-69.462,-176.669,7.526,148.462
C02496=1191.636,300.093,-69.432,-176.672,7.523,148.463
C02497=1191.641,299.845,-69.402,-176.675,7.520,148.463
C02498=1191.645,299.597,-69.372,-176.677,7.517,148.463
C02499=1191.649,299.349,-69.343,-176.679,7.514,148.463
C02500=1191.654,299.101,-69.312,-176.682,7.511,148.462
C02501=1191.658,298.853,-69.282,-176.684,7.508,148.462
C02502=1191.662,298.604,-69.253,-176.687,7.505,148.462
C02503=1191.666,298.356,-69.224,-176.689,7.503,148.463
C02504=1191.671,298.108,-69.193,-176.692,7.500,148.463
C02505=1191.675,297.860,-69.163,-176.695,7.497,148.463
C02506=1191.679,297.612,-69.134,-176.697,7.494,148.463
C02507=1191.684,297.363,-69.104,-176.700,7.492,148.463
C02508=1191.687,297.116,-69.074,-176.702,7.489,148.463
C02509=1191.692,296.867,-69.044,-176.705,7.486,148.463
C02510=1191.697,296.619,-69.015,-176.707,7.484,148.463
C02511=1191.701,296.371,-68.985,-176.710,7.481,148.463
C02512=1191.705,296.122,-68.956,-176.713,7.478,148.463
C02513=1191.709,295.874,-68.926,-176.715,7.475,148.463
C02514=1191.713,295.626,-68.896,-176.717,7.472,148.463
C02515=1191.718,295.378,-68.866,-176.720,7.469,148.463
C02516=1191.722,295.130,-68.837,-176.723,7.466,148.463
C02517=1191.726,294.881,-68.807,-176.725,7.464,148.463
C02518=1191.730,294.633,-68.778,-176.728,7.461,148.463
C02519=1191.735,294.385,-68.748,-176.730,7.458,148.463
C02520=1191.739,294.136,-68.719,-176.733,7.455,148.463
C02521=1191.743,293.888,-68.689,-176.735,7.453,148.463
C02522=1191.747,293.640,-68.660,-176.737,7.450,148.463
C02523=1191.752,293.392,-68.631,-176.740,7.447,148.463
C02524=1191.757,293.144,-68.601,-176.742,7.445,148.463
C02525=1191.761,292.895,-68.571,-176.745,7.441,148.463
C02526=1191.765,292.647,-68.542,-176.748,7.438,148.463
C02527=1191.769,292.399,-68.512,-176.750,7.436,148.463
C02528=1191.774,292.151,-68.483,-176.753,7.433,148.463
C02529=1191.778,291.902,-68.454,-176.755,7.430,148.463
C02530=1191.782,291.654,-68.424,-176.758,7.427,148.463
C02531=1191.786,291.406,-68.395,-176.760,7.425,148.463
C02532=1191.791,291.158,-68.366,-176.763,7.422,148.463
C02533=1191.795,290.910,-68.336,-176.766,7.419,148.463
C02534=1191.799,290.662,-68.307,-176.768,7.417,148.463
C02535=1191.804,290.413,-68.278,-176.770,7.414,148.463
C02536=1191.808,290.165,-68.249,-176.774,7.411,148.464
C02537=1191.812,289.916,-68.219,-176.776,7.409,148.464
C02538=1191.816,289.668,-68.190,-176.778,7.406,148.464
C02539=1191.821,289.421,-68.161,-176.781,7.403,148.464
C02540=1191.826,289.172,-68.132,-176.783,7.401,148.464
C02541=1191.829,288.897,-68.099,-176.786,7.398,148.464
C02542=1191.834,288.623,-68.067,-176.789,7.394,148.464
C02543=1191.840,288.349,-68.034,-176.792,7.391,148.464
C02544=1191.844,288.074,-68.002,-176.795,7.388,148.464
C02545=1191.849,287.826,-67.973,-176.797,7.386,148.464
C02546=1191.853,287.577,-67.945,-176.800,7.383,148.464
C02547=1191.857,287.329,-67.915,-176.802,7.380,148.464
C02548=1191.861,287.081,-67.886,-176.804,7.378,148.464
C02549=1191.866,286.832,-67.857,-176.808,7.375,148.464
C02550=1191.870,286.585,-67.828,-176.810,7.372,148.464
C02551=1191.874,286.336,-67.799,-176.813,7.370,148.465
C02552=1191.879,286.087,-67.770,-176.815,7.367,148.465
C02553=1191.883,285.839,-67.741,-176.818,7.364,148.465
C02554=1191.888,285.592,-67.712,-176.820,7.362,148.465
C02555=1191.892,285.343,-67.683,-176.823,7.359,148.465
C02556=1191.895,285.095,-67.654,-176.826,7.356,148.465
C02557=1191.900,284.846,-67.625,-176.828,7.353,148.465
C02558=1191.905,284.598,-67.596,-176.830,7.350,148.465
C02559=1191.909,284.350,-67.567,-176.833,7.347,148.465
C02560=1191.913,284.101,-67.538,-176.835,7.345,148.465
C02561=1191.917,283.854,-67.510,-176.838,7.342,148.465
C02562=1191.922,283.605,-67.481,-176.841,7.340,148.465
C02563=1191.926,283.357,-67.451,-176.843,7.337,148.465
C02564=1191.931,283.108,-67.423,-176.846,7.334,148.465
C02565=1191.935,282.861,-67.394,-176.848,7.332,148.465
C02566=1191.939,282.612,-67.365,-176.851,7.329,148.465
C02567=1191.943,282.363,-67.336,-176.854,7.326,148.465
C02568=1191.948,282.115,-67.308,-176.856,7.324,148.466
C02569=1191.952,281.867,-67.280,-176.858,7.321,148.466
C02570=1191.956,281.618,-67.250,-176.861,7.318,148.466
C02571=1191.961,281.370,-67.222,-176.863,7.316,148.466
C02572=1191.965,281.122,-67.193,-176.866,7.313,148.466
C02573=1191.969,280.873,-67.164,-176.869,7.310,148.466
C02574=1191.974,280.625,-67.136,-176.871,7.308,148.466
C02575=1191.978,280.377,-67.107,-176.874,7.305,148.466
C02576=1191.982,280.128,-67.078,-176.876,7.303,148.466
C02577=1191.987,279.880,-67.050,-176.879,7.300,148.466
C02578=1191.991,279.632,-67.021,-176.882,7.297,148.466
C02579=1191.995,279.383,-66.992,-176.884,7.295,148.466
C02580=1192.000,279.135,-66.964,-176.887,7.292,148.467
C02581=1192.004,278.887,-66.935,-176.889,7.290,148.467
C02582=1192.009,278.639,-66.907,-176.892,7.287,148.467
C02583=1192.013,278.390,-66.878,-176.895,7.284,148.467
C02584=1192.017,278.142,-66.850,-176.897,7.282,148.467
C02585=1192.021,277.894,-66.821,-176.899,7.279,148.467
C02586=1192.026,277.645,-66.792,-176.902,7.276,148.467
C02587=1192.031,277.397,-66.764,-176.905,7.274,148.467
C02588=1192.035,277.149,-66.736,-176.907,7.271,148.467
C02589=1192.039,276.900,-66.707,-176.910,7.269,148.467
C02590=1192.043,276.652,-66.679,-176.912,7.266,148.467
C02591=1192.048,276.404,-66.650,-176.915,7.263,148.467
C02592=1192.052,276.156,-66.622,-176.917,7.261,148.467
C02593=1192.056,275.907,-66.593,-176.920,7.258,148.468
C02594=1192.061,275.659,-66.566,-176.923,7.256,148.468
C02595=1192.065,275.410,-66.537,-176.925,7.253,148.468
C02596=1192.069,275.161,-66.509,-176.928,7.250,148.468
C02597=1192.074,274.913,-66.480,-176.930,7.247,148.468
C02598=1192.078,274.665,-66.452,-176.933,7.244,148.468
C02599=1192.083,274.417,-66.423,-176.935,7.243,148.468
C02600=1192.086,274.169,-66.395,-176.938,7.240,148.468
C02601=1192.091,273.921,-66.367,-176.940,7.237,148.468
C02602=1192.095,273.672,-66.339,-176.943,7.234,148.468
C02603=1192.100,273.424,-66.311,-176.946,7.231,148.468
C02604=1192.104,273.175,-66.282,-176.948,7.230,148.469
C02605=1192.108,272.927,-66.254,-176.951,7.227,148.469
C02606=1192.113,272.678,-66.226,-176.953,7.224,148.469
C02607=1192.117,272.430,-66.198,-176.956,7.221,148.469
C02608=1192.121,272.181,-66.170,-176.959,7.218,148.469
C02609=1192.126,271.933,-66.142,-176.961,7.217,148.469
C02610=1192.130,271.684,-66.114,-176.964,7.214,148.469
C02611=1192.135,271.437,-66.086,-176.966,7.211,148.469
C02612=1192.139,271.188,-66.057,-176.969,7.208,148.469
C02613=1192.143,270.940,-66.029,-176.971,7.207,148.470
C02614=1192.148,270.691,-66.001,-176.974,7.204,148.470
C02615=1192.152,270.443,-65.973,-176.977,7.201,148.470
C02616=1192.157,270.195,-65.945,-176.979,7.198,148.470
C02617=1192.161,269.946,-65.917,-176.982,7.195,148.470
C02618=1192.166,269.698,-65.889,-176.984,7.194,148.470
C02619=1192.169,269.449,-65.861,-176.987,7.191,148.470
C02620=1192.174,269.201,-65.833,-176.989,7.188,148.470
C02621=1192.178,268.952,-65.805,-176.992,7.185,148.470
C02622=1192.183,268.704,-65.778,-176.995,7.184,148.471
C02623=1192.187,268.456,-65.750,-176.997,7.181,148.471
C02624=1192.192,268.207,-65.721,-177.000,7.178,148.471
C02625=1192.196,267.959,-65.693,-177.002,7.175,148.471
C02626=1192.200,267.710,-65.666,-177.005,7.173,148.471
C02627=1192.205,267.462,-65.638,-177.008,7.171,148.471
C02628=1192.210,267.214,-65.610,-177.010,7.168,148.471
C02629=1192.214,266.965,-65.582,-177.012,7.165,148.471
C02630=1192.218,266.717,-65.555,-177.016,7.163,148.472
C02631=1192.222,266.468,-65.526,-177.018,7.161,148.472
C02632=1192.226,266.220,-65.499,-177.020,7.158,148.472
C02633=1192.232,265.972,-65.471,-177.023,7.155,148.472
C02634=1192.235,265.723,-65.443,-177.026,7.153,148.472
C02635=1192.240,265.475,-65.416,-177.028,7.151,148.472
C02636=1192.244,265.227,-65.388,-177.031,7.148,148.472
C02637=1192.248,264.978,-65.361,-177.033,7.145,148.472
C02638=1192.253,264.730,-65.333,-177.036,7.143,148.473
C02639=1192.258,264.482,-65.304,-177.038,7.141,148.473
C02640=1192.262,264.232,-65.277,-177.041,7.138,148.473
C02641=1192.266,263.984,-65.249,-177.044,7.135,148.473
C02642=1192.271,263.736,-65.222,-177.046,7.133,148.473
C02643=1192.275,263.487,-65.194,-177.049,7.130,148.473
C02644=1192.279,263.239,-65.167,-177.051,7.128,148.473
C02645=1192.285,262.966,-65.137,-177.054,7.125,148.473
C02646=1192.289,262.693,-65.106,-177.057,7.122,148.473
C02647=1192.294,262.421,-65.076,-177.060,7.119,148.474
C02648=1192.298,262.147,-65.046,-177.062,7.117,148.474
C02649=1192.303,261.899,-65.019,-177.065,7.114,148.474
C02650=1192.307,261.651,-64.991,-177.068,7.112,148.474
C02651=1192.312,261.402,-64.964,-177.070,7.109,148.474
C02652=1192.316,261.154,-64.936,-177.073,7.107,148.474
C02653=1192.320,260.905,-64.909,-177.076,7.104,148.475
C02654=1192.325,260.657,-64.881,-177.078,7.102,148.475
C02655=1192.329,260.409,-64.854,-177.081,7.099,148.475
C02656=1192.334,260.160,-64.826,-177.083,7.097,148.475
C02657=1192.338,259.912,-64.798,-177.086,7.094,148.475
C02658=1192.343,259.663,-64.771,-177.088,7.092,148.475
C02659=1192.347,259.415,-64.744,-177.091,7.090,148.475
C02660=1192.351,259.166,-64.717,-177.094,7.087,148.475
C02661=1192.356,258.918,-64.689,-177.096,7.084,148.476
C02662=1192.360,258.669,-64.662,-177.099,7.083,148.476
C02663=1192.365,258.421,-64.635,-177.102,7.080,148.476
C02664=1192.369,258.172,-64.607,-177.104,7.077,148.476
C02665=1192.373,257.924,-64.580,-177.107,7.075,148.476
C02666=1192.378,257.675,-64.553,-177.109,7.073,148.476
C02667=1192.383,257.427,-64.526,-177.112,7.070,148.476
C02668=1192.387,257.178,-64.499,-177.114,7.068,148.477
C02669=1192.391,256.930,-64.470,-177.117,7.065,148.477
C02670=1192.395,256.682,-64.444,-177.119,7.063,148.477
C02671=1192.400,256.433,-64.417,-177.123,7.060,148.477
C02672=1192.404,256.185,-64.390,-177.125,7.058,148.477
C02673=1192.409,255.936,-64.363,-177.127,7.056,148.477
C02674=1192.414,255.688,-64.336,-177.130,7.053,148.478
C02675=1192.418,255.438,-64.308,-177.132,7.051,148.478
C02676=1192.422,255.190,-64.281,-177.135,7.048,148.478
C02677=1192.426,254.942,-64.254,-177.138,7.046,148.478
C02678=1192.431,254.694,-64.227,-177.140,7.043,148.478
C02679=1192.435,254.445,-64.200,-177.143,7.041,148.478
C02680=1192.440,254.197,-64.173,-177.146,7.038,148.478
C02681=1192.445,253.948,-64.146,-177.148,7.036,148.479
C02682=1192.449,253.699,-64.118,-177.151,7.033,148.479
C02683=1192.453,253.451,-64.092,-177.153,7.031,148.479
C02684=1192.457,253.202,-64.065,-177.156,7.029,148.479
C02685=1192.462,252.954,-64.038,-177.159,7.026,148.479
C02686=1192.466,252.705,-64.011,-177.161,7.024,148.479
C02687=1192.470,252.457,-63.984,-177.164,7.021,148.480
C02688=1192.475,252.209,-63.957,-177.166,7.019,148.480
C02689=1192.480,251.960,-63.930,-177.169,7.017,148.480
C02690=1192.484,251.712,-63.903,-177.171,7.014,148.480
C02691=1192.488,251.464,-63.877,-177.174,7.012,148.480
C02692=1192.492,251.214,-63.849,-177.177,7.010,148.480
C02693=1192.497,250.966,-63.822,-177.179,7.007,148.481
C02694=1192.501,250.717,-63.796,-177.182,7.005,148.481
C02695=1192.506,250.469,-63.769,-177.184,7.003,148.481
C02696=1192.511,250.220,-63.742,-177.187,7.000,148.481
C02697=1192.515,249.972,-63.715,-177.190,6.998,148.481
C02698=1192.519,249.723,-63.689,-177.192,6.996,148.481
C02699=1192.524,249.475,-63.662,-177.195,6.993,148.482
C02700=1192.528,249.227,-63.635,-177.197,6.991,148.482
C02701=1192.533,248.978,-63.609,-177.200,6.988,148.482
C02702=1192.537,248.729,-63.582,-177.202,6.986,148.482
C02703=1192.541,248.481,-63.555,-177.205,6.984,148.482
C02704=1192.546,248.232,-63.528,-177.208,6.981,148.482
C02705=1192.551,247.983,-63.502,-177.210,6.979,148.483
C02706=1192.555,247.735,-63.476,-177.213,6.976,148.483
C02707=1192.559,247.487,-63.448,-177.215,6.974,148.483
C02708=1192.563,247.238,-63.422,-177.218,6.972,148.483
C02709=1192.568,246.989,-63.396,-177.221,6.969,148.483
C02710=1192.573,246.741,-63.369,-177.223,6.968,148.484
C02711=1192.577,246.493,-63.342,-177.226,6.965,148.484
C02712=1192.582,246.244,-63.316,-177.228,6.962,148.484
C02713=1192.586,245.995,-63.289,-177.231,6.961,148.484
C02714=1192.590,245.747,-63.262,-177.234,6.958,148.484
C02715=1192.595,245.498,-63.236,-177.236,6.956,148.484
C02716=1192.599,245.250,-63.209,-177.239,6.953,148.485
C02717=1192.603,245.001,-63.183,-177.242,6.951,148.485
C02718=1192.608,244.752,-63.157,-177.244,6.949,148.485
C02719=1192.612,244.504,-63.130,-177.247,6.946,148.485
C02720=1192.617,244.255,-63.104,-177.249,6.944,148.485
C02721=1192.621,244.007,-63.077,-177.252,6.942,148.486
C02722=1192.626,243.758,-63.051,-177.254,6.939,148.486
C02723=1192.630,243.509,-63.025,-177.257,6.937,148.486
C02724=1192.635,243.262,-62.998,-177.260,6.934,148.486
C02725=1192.639,243.013,-62.972,-177.262,6.932,148.486
C02726=1192.644,242.764,-62.945,-177.265,6.930,148.486
C02727=1192.648,242.516,-62.919,-177.268,6.928,148.487
C02728=1192.653,242.267,-62.892,-177.270,6.925,148.487
C02729=1192.657,242.018,-62.866,-177.273,6.924,148.487
C02730=1192.661,241.769,-62.841,-177.275,6.921,148.487
C02731=1192.666,241.521,-62.814,-177.278,6.919,148.488
C02732=1192.670,241.272,-62.788,-177.280,6.917,148.488
C02733=1192.675,241.024,-62.761,-177.283,6.914,148.488
C02734=1192.680,240.776,-62.735,-177.286,6.912,148.488
C02735=1192.684,240.527,-62.709,-177.289,6.909,148.488
C02736=1192.689,240.278,-62.683,-177.291,6.907,148.488
C02737=1192.693,240.029,-62.657,-177.294,6.905,148.489
C02738=1192.697,239.781,-62.630,-177.296,6.902,148.489
C02739=1192.702,239.532,-62.604,-177.299,6.900,148.489
C02740=1192.706,239.283,-62.578,-177.301,6.898,148.489
C02741=1192.710,239.036,-62.552,-177.304,6.896,148.490
C02742=1192.715,238.787,-62.526,-177.306,6.893,148.490
C02743=1192.720,238.538,-62.500,-177.309,6.892,148.490
C02744=1192.724,238.290,-62.474,-177.312,6.889,148.490
C02745=1192.728,238.041,-62.447,-177.314,6.887,148.490
C02746=1192.733,237.793,-62.422,-177.317,6.885,148.490
C02747=1192.738,237.544,-62.396,-177.320,6.882,148.491
C02748=1192.742,237.295,-62.369,-177.322,6.880,148.491
C02749=1192.747,237.023,-62.341,-177.325,6.877,148.491
C02750=1192.751,236.752,-62.312,-177.328,6.875,148.491
C02751=1192.757,236.481,-62.285,-177.331,6.872,148.491
C02752=1192.761,236.209,-62.257,-177.333,6.870,148.492
C02753=1192.766,235.960,-62.230,-177.336,6.868,148.492
C02754=1192.770,235.712,-62.204,-177.339,6.866,148.492
C02755=1192.775,235.464,-62.178,-177.341,6.864,148.493
C02756=1192.779,235.215,-62.153,-177.344,6.861,148.493
C02757=1192.784,234.966,-62.126,-177.347,6.859,148.493
C02758=1192.788,234.717,-62.101,-177.349,6.857,148.493
C02759=1192.793,234.469,-62.075,-177.352,6.854,148.493
C02760=1192.797,234.221,-62.049,-177.355,6.852,148.494
C02761=1192.801,233.972,-62.023,-177.357,6.850,148.494
C02762=1192.806,233.723,-61.997,-177.360,6.848,148.494
C02763=1192.811,233.475,-61.971,-177.362,6.845,148.494
C02764=1192.815,233.226,-61.945,-177.365,6.844,148.494
C02765=1192.820,232.977,-61.920,-177.368,6.841,148.495
C02766=1192.824,232.729,-61.894,-177.370,6.839,148.495
C02767=1192.829,232.480,-61.869,-177.373,6.837,148.495
C02768=1192.833,232.231,-61.843,-177.375,6.835,148.495
C02769=1192.837,231.982,-61.817,-177.378,6.832,148.496
C02770=1192.842,231.734,-61.792,-177.381,6.830,148.496
C02771=1192.847,231.485,-61.765,-177.383,6.828,148.496
C02772=1192.851,231.236,-61.740,-177.386,6.825,148.496
C02773=1192.856,230.988,-61.714,-177.388,6.823,148.496
C02774=1192.860,230.739,-61.688,-177.391,6.821,148.497
C02775=1192.864,230.491,-61.663,-177.394,6.820,148.497
C02776=1192.870,230.242,-61.638,-177.396,6.817,148.497
C02777=1192.874,229.993,-61.612,-177.399,6.815,148.497
C02778=1192.878,229.744,-61.587,-177.401,6.813,148.498
C02779=1192.883,229.496,-61.561,-177.404,6.810,148.498
C02780=1192.887,229.247,-61.535,-177.407,6.808,148.498
C02781=1192.891,228.999,-61.510,-177.409,6.806,148.498
C02782=1192.896,228.751,-61.484,-177.412,6.804,148.499
C02783=1192.900,228.502,-61.459,-177.415,6.801,148.499
C02784=1192.905,228.252,-61.433,-177.417,6.799,148.499
C02785=1192.910,228.004,-61.408,-177.420,6.798,148.499
C02786=1192.914,227.755,-61.382,-177.422,6.795,148.499
C02787=1192.919,227.507,-61.357,-177.425,6.793,148.500
C02788=1192.923,227.258,-61.332,-177.428,6.791,148.500
C02789=1192.927,227.009,-61.306,-177.430,6.789,148.500
C02790=1192.932,226.761,-61.281,-177.433,6.786,148.500
C02791=1192.937,226.512,-61.255,-177.436,6.784,148.501
C02792=1192.942,226.263,-61.230,-177.438,6.782,148.501
C02793=1192.946,226.015,-61.205,-177.441,6.780,148.501
C02794=1192.950,225.766,-61.179,-177.444,6.778,148.501
C02795=1192.954,225.518,-61.154,-177.446,6.776,148.502
C02796=1192.959,225.269,-61.129,-177.449,6.774,148.502
C02797=1192.964,225.021,-61.104,-177.451,6.772,148.502
C02798=1192.968,224.772,-61.078,-177.454,6.769,148.502
C02799=1192.972,224.522,-61.053,-177.457,6.767,148.503
C02800=1192.977,224.274,-61.027,-177.459,6.765,148.503
C02801=1192.982,224.025,-61.002,-177.462,6.763,148.503
C02802=1192.986,223.777,-60.977,-177.465,6.760,148.503
C02803=1192.990,223.528,-60.952,-177.467,6.759,148.504
C02804=1192.995,223.279,-60.927,-177.470,6.757,148.504
C02805=1192.999,223.031,-60.901,-177.472,6.755,148.504
C02806=1193.004,222.782,-60.877,-177.475,6.753,148.504
C02807=1193.009,222.533,-60.851,-177.478,6.750,148.505
C02808=1193.014,222.284,-60.826,-177.480,6.748,148.505
C02809=1193.017,222.036,-60.801,-177.483,6.746,148.505
C02810=1193.022,221.787,-60.777,-177.485,6.744,148.505
C02811=1193.027,221.538,-60.751,-177.488,6.741,148.506
C02812=1193.032,221.290,-60.726,-177.491,6.740,148.506
C02813=1193.035,221.041,-60.701,-177.493,6.737,148.506
C02814=1193.040,220.792,-60.676,-177.496,6.736,148.506
C02815=1193.045,220.544,-60.651,-177.499,6.733,148.507
C02816=1193.050,220.295,-60.626,-177.501,6.731,148.507
C02817=1193.053,220.046,-60.601,-177.504,6.729,148.507
C02818=1193.058,219.798,-60.576,-177.506,6.727,148.507
C02819=1193.063,219.549,-60.550,-177.509,6.725,148.508
C02820=1193.068,219.300,-60.526,-177.512,6.722,148.508
C02821=1193.072,219.051,-60.501,-177.514,6.721,148.508
C02822=1193.076,218.803,-60.476,-177.517,6.719,148.509
C02823=1193.081,218.553,-60.451,-177.519,6.717,148.509
C02824=1193.085,218.305,-60.427,-177.522,6.714,148.509
C02825=1193.090,218.057,-60.401,-177.525,6.712,148.509
C02826=1193.095,217.808,-60.376,-177.528,6.710,148.510
C02827=1193.099,217.559,-60.352,-177.530,6.708,148.510
C02828=1193.103,217.310,-60.326,-177.533,6.706,148.510
C02829=1193.108,217.062,-60.302,-177.536,6.704,148.510
C02830=1193.112,216.812,-60.277,-177.538,6.702,148.511
C02831=1193.117,216.564,-60.252,-177.541,6.700,148.511
C02832=1193.122,216.316,-60.227,-177.543,6.698,148.511
C02833=1193.126,216.067,-60.203,-177.546,6.696,148.512
C02834=1193.131,215.818,-60.178,-177.549,6.693,148.512
C02835=1193.135,215.569,-60.153,-177.551,6.691,148.512
C02836=1193.140,215.321,-60.128,-177.554,6.690,148.512
C02837=1193.145,215.072,-60.104,-177.557,6.688,148.513
C02838=1193.149,214.823,-60.079,-177.559,6.686,148.513
C02839=1193.154,214.574,-60.055,-177.562,6.683,148.513
C02840=1193.158,214.326,-60.030,-177.565,6.681,148.513
C02841=1193.162,214.077,-60.005,-177.567,6.679,148.514
C02842=1193.167,213.828,-59.981,-177.570,6.677,148.514
C02843=1193.171,213.579,-59.956,-177.572,6.675,148.514
C02844=1193.176,213.331,-59.932,-177.575,6.673,148.514
C02845=1193.181,213.082,-59.907,-177.578,6.671,148.515
C02846=1193.185,212.833,-59.882,-177.581,6.669,148.515
C02847=1193.190,212.584,-59.858,-177.583,6.667,148.515
C02848=1193.194,212.336,-59.834,-177.585,6.665,148.516
C02849=1193.198,212.087,-59.808,-177.588,6.663,148.516
C02850=1193.203,211.838,-59.784,-177.591,6.661,148.516
C02851=1193.208,211.590,-59.759,-177.594,6.658,148.516
C02852=1193.212,211.341,-59.735,-177.596,6.657,148.517
C02853=1193.217,211.070,-59.709,-177.599,6.655,148.517
C02854=1193.222,210.800,-59.682,-177.602,6.652,148.517
C02855=1193.227,210.529,-59.655,-177.605,6.650,148.518
C02856=1193.232,210.259,-59.628,-177.608,6.648,148.518
C02857=1193.236,210.010,-59.604,-177.611,6.646,148.518
C02858=1193.241,209.761,-59.580,-177.613,6.644,148.518
C02859=1193.246,209.513,-59.555,-177.615,6.642,148.519
C02860=1193.250,209.264,-59.531,-177.618,6.640,148.519
C02861=1193.255,209.015,-59.506,-177.621,6.637,148.519
C02862=1193.260,208.766,-59.483,-177.624,6.636,148.520
C02863=1193.265,208.517,-59.458,-177.626,6.634,148.520
C02864=1193.268,208.268,-59.434,-177.629,6.632,148.520
C02865=1193.273,208.020,-59.410,-177.631,6.630,148.521
C02866=1193.278,207.771,-59.385,-177.634,6.628,148.521
C02867=1193.282,207.523,-59.361,-177.637,6.626,148.521
C02868=1193.286,207.274,-59.337,-177.639,6.623,148.521
C02869=1193.291,207.025,-59.312,-177.642,6.622,148.522
C02870=1193.296,206.776,-59.289,-177.645,6.620,148.522
C02871=1193.300,206.527,-59.265,-177.647,6.618,148.522
C02872=1193.306,206.279,-59.240,-177.650,6.616,148.523
C02873=1193.309,206.030,-59.215,-177.653,6.614,148.523
C02874=1193.314,205.781,-59.192,-177.655,6.612,148.523
C02875=1193.319,205.532,-59.167,-177.658,6.609,148.523
C02876=1193.324,205.283,-59.143,-177.661,6.608,148.524
C02877=1193.328,205.035,-59.119,-177.663,6.606,148.524
C02878=1193.333,204.785,-59.095,-177.666,6.604,148.524
C02879=1193.337,204.537,-59.071,-177.668,6.602,148.525
C02880=1193.342,204.288,-59.047,-177.671,6.600,148.525
C02881=1193.346,204.040,-59.023,-177.674,6.598,148.525
C02882=1193.351,203.790,-58.999,-177.676,6.596,148.526
C02883=1193.356,203.542,-58.975,-177.679,6.594,148.526
C02884=1193.360,203.293,-58.950,-177.682,6.592,148.526
C02885=1193.364,203.044,-58.927,-177.684,6.590,148.526
C02886=1193.369,202.795,-58.903,-177.687,6.588,148.527
C02887=1193.374,202.547,-58.878,-177.690,6.586,148.527
C02888=1193.378,202.298,-58.855,-177.692,6.584,148.527
C02889=1193.383,202.049,-58.831,-177.695,6.583,148.528
C02890=1193.388,201.800,-58.807,-177.698,6.581,148.528
C02891=1193.391,201.551,-58.783,-177.700,6.579,148.528
C02892=1193.396,201.302,-58.760,-177.703,6.576,148.529
C02893=1193.401,201.053,-58.735,-177.706,6.574,148.529
C02894=1193.406,200.805,-58.711,-177.708,6.572,148.529
C02895=1193.410,200.556,-58.687,-177.711,6.571,148.530
C02896=1193.415,200.308,-58.663,-177.714,6.569,148.530
C02897=1193.419,200.058,-58.640,-177.716,6.567,148.530
C02898=1193.424,199.810,-58.616,-177.718,6.565,148.530
C02899=1193.428,199.561,-58.593,-177.721,6.563,148.531
C02900=1193.432,199.312,-58.568,-177.724,6.561,148.531
C02901=1193.438,199.063,-58.544,-177.726,6.559,148.531
C02902=1193.442,198.814,-58.520,-177.729,6.558,148.532
C02903=1193.447,198.565,-58.497,-177.732,6.555,148.532
C02904=1193.452,198.316,-58.473,-177.735,6.553,148.532
C02905=1193.456,198.068,-58.449,-177.737,6.551,148.533
C02906=1193.461,197.819,-58.426,-177.740,6.549,148.533
C02907=1193.465,197.570,-58.402,-177.742,6.547,148.533
C02908=1193.470,197.321,-58.379,-177.745,6.546,148.534
C02909=1193.474,197.072,-58.355,-177.748,6.544,148.534
C02910=1193.479,196.824,-58.331,-177.750,6.542,148.534
C02911=1193.483,196.575,-58.308,-177.753,6.540,148.535
C02912=1193.488,196.326,-58.284,-177.756,6.538,148.535
C02913=1193.493,196.077,-58.260,-177.758,6.536,148.535
C02914=1193.497,195.828,-58.237,-177.761,6.534,148.535
C02915=1193.502,195.579,-58.214,-177.763,6.533,148.536
C02916=1193.506,195.331,-58.190,-177.766,6.530,148.536
C02917=1193.511,195.082,-58.166,-177.769,6.528,148.536
C02918=1193.516,194.833,-58.143,-177.772,6.526,148.537
C02919=1193.520,194.584,-58.119,-177.774,6.525,148.537
C02920=1193.525,194.335,-58.095,-177.777,6.523,148.538
C02921=1193.530,194.086,-58.072,-177.780,6.521,148.538
C02922=1193.534,193.837,-58.049,-177.782,6.519,148.538
C02923=1193.539,193.589,-58.025,-177.785,6.517,148.538
C02924=1193.543,193.340,-58.001,-177.787,6.515,148.539
C02925=1193.548,193.091,-57.978,-177.790,6.513,148.539
C02926=1193.552,192.842,-57.955,-177.793,6.512,148.539
C02927=1193.557,192.593,-57.932,-177.795,6.510,148.540
C02928=1193.561,192.344,-57.908,-177.798,6.508,148.540
C02929=1193.566,192.096,-57.884,-177.801,6.506,148.540
C02930=1193.571,191.847,-57.861,-177.803,6.504,148.541
C02931=1193.575,191.598,-57.838,-177.806,6.503,148.541
C02932=1193.580,191.348,-57.814,-177.809,6.501,148.542
C02933=1193.585,191.100,-57.791,-177.811,6.499,148.542
C02934=1193.590,190.851,-57.768,-177.813,6.497,148.542
C02935=1193.594,190.602,-57.745,-177.816,6.495,148.542
C02936=1193.599,190.353,-57.722,-177.819,6.493,148.543
C02937=1193.603,190.104,-57.698,-177.821,6.491,148.543
C02938=1193.608,189.855,-57.675,-177.824,6.490,148.543
C02939=1193.613,189.606,-57.652,-177.827,6.488,148.544
C02940=1193.616,189.358,-57.628,-177.830,6.485,148.544
C02941=1193.621,189.109,-57.605,-177.833,6.483,148.544
C02942=1193.626,188.860,-57.581,-177.835,6.482,148.545
C02943=1193.631,188.612,-57.558,-177.838,6.480,148.545
C02944=1193.636,188.363,-57.535,-177.841,6.478,148.545
C02945=1193.640,188.114,-57.512,-177.843,6.476,148.546
C02946=1193.645,187.864,-57.490,-177.846,6.474,148.546
C02947=1193.649,187.615,-57.466,-177.849,6.473,148.547
C02948=1193.654,187.366,-57.443,-177.851,6.471,148.547
C02949=1193.658,187.118,-57.420,-177.853,6.469,148.547
C02950=1193.663,186.869,-57.397,-177.856,6.467,148.547
C02951=1193.668,186.620,-57.374,-177.859,6.465,148.548
C02952=1193.673,186.371,-57.351,-177.861,6.463,148.548
C02953=1193.677,186.122,-57.328,-177.864,6.461,148.548
C02954=1193.681,185.873,-57.304,-177.867,6.460,148.549
C02955=1193.686,185.624,-57.281,-177.869,6.458,148.549
C02956=1193.691,185.376,-57.259,-177.872,6.456,148.550
C02957=1193.696,185.107,-57.234,-177.875,6.454,148.550
C02958=1193.701,184.837,-57.209,-177.877,6.452,148.550
C02959=1193.706,184.567,-57.184,-177.881,6.451,148.551
C02960=1193.711,184.298,-57.159,-177.884,6.448,148.551
C02961=1193.715,184.049,-57.136,-177.886,6.447,148.551
C02962=1193.720,183.799,-57.114,-177.889,6.445,148.552
C02963=1193.725,183.550,-57.090,-177.892,6.443,148.552
C02964=1193.729,183.301,-57.068,-177.894,6.441,148.553
C02965=1193.734,183.053,-57.045,-177.897,6.440,148.553
C02966=1193.739,182.804,-57.022,-177.899,6.438,148.553
C02967=1193.743,182.555,-56.999,-177.901,6.436,148.553
C02968=1193.748,182.306,-56.976,-177.904,6.434,148.554
C02969=1193.752,182.058,-56.953,-177.907,6.433,148.554
C02970=1193.757,181.808,-56.931,-177.909,6.431,148.554
C02971=1193.761,181.559,-56.908,-177.912,6.429,148.555
C02972=1193.766,181.310,-56.885,-177.915,6.427,148.555
C02973=1193.772,181.061,-56.862,-177.917,6.425,148.556
C02974=1193.776,180.813,-56.840,-177.920,6.424,148.556
C02975=1193.780,180.564,-56.816,-177.923,6.422,148.556
C02976=1193.785,180.314,-56.794,-177.925,6.420,148.557
C02977=1193.790,180.066,-56.771,-177.928,6.418,148.557
C02978=1193.794,179.817,-56.748,-177.931,6.417,148.557
C02979=1193.799,179.568,-56.726,-177.933,6.415,148.558
C02980=1193.803,179.319,-56.703,-177.936,6.413,148.558
C02981=1193.808,179.070,-56.681,-177.939,6.411,148.558
C02982=1193.812,178.821,-56.658,-177.941,6.409,148.559
C02983=1193.817,178.572,-56.635,-177.944,6.408,148.559
C02984=1193.822,178.324,-56.613,-177.947,6.406,148.560
C02985=1193.827,178.074,-56.590,-177.949,6.404,148.560
C02986=1193.831,177.825,-56.568,-177.952,6.402,148.560
C02987=1193.836,177.577,-56.545,-177.955,6.400,148.561
C02988=1193.841,177.327,-56.523,-177.957,6.399,148.561
C02989=1193.845,177.078,-56.500,-177.959,6.398,148.561
C02990=1193.850,176.830,-56.477,-177.962,6.396,148.562
C02991=1193.854,176.580,-56.455,-177.965,6.394,148.562
C02992=1193.859,176.331,-56.432,-177.967,6.392,148.562
C02993=1193.864,176.083,-56.410,-177.970,6.390,148.563
C02994=1193.868,175.834,-56.388,-177.973,6.389,148.563
C02995=1193.873,175.584,-56.365,-177.976,6.387,148.564
C02996=1193.877,175.336,-56.343,-177.979,6.385,148.564
C02997=1193.882,175.087,-56.320,-177.981,6.384,148.564
C02998=1193.887,174.838,-56.298,-177.984,6.382,148.565
C02999=1193.891,174.589,-56.275,-177.987,6.380,148.565
C03000=1193.896,174.340,-56.253,-177.989,6.378,148.566
C03001=1193.901,174.092,-56.230,-177.992,6.376,148.566
C03002=1193.905,173.842,-56.208,-177.995,6.375,148.566
C03003=1193.910,173.593,-56.186,-177.997,6.374,148.567
C03004=1193.915,173.345,-56.163,-177.999,6.372,148.567
C03005=1193.919,173.095,-56.141,-178.002,6.370,148.567
C03006=1193.925,172.846,-56.119,-178.005,6.368,148.568
C03007=1193.929,172.597,-56.097,-178.007,6.366,148.568
C03008=1193.933,172.349,-56.075,-178.010,6.365,148.568
C03009=1193.938,172.099,-56.052,-178.013,6.363,148.569
C03010=1193.943,171.850,-56.030,-178.015,6.361,148.569
C03011=1193.948,171.601,-56.008,-178.018,6.359,148.570
C03012=1193.951,171.353,-55.985,-178.021,6.358,148.570
C03013=1193.957,171.104,-55.963,-178.023,6.357,148.570
C03014=1193.961,170.854,-55.941,-178.026,6.355,148.571
C03015=1193.966,170.606,-55.919,-178.028,6.353,148.571
C03016=1193.970,170.357,-55.897,-178.031,6.351,148.571
C03017=1193.976,170.108,-55.874,-178.034,6.350,148.572
C03018=1193.980,169.859,-55.852,-178.037,6.348,148.572
C03019=1193.985,169.610,-55.831,-178.039,6.346,148.573
C03020=1193.989,169.361,-55.809,-178.042,6.344,148.573
C03021=1193.994,169.111,-55.786,-178.045,6.343,148.573
C03022=1193.999,168.863,-55.764,-178.047,6.342,148.574
C03023=1194.003,168.614,-55.742,-178.050,6.340,148.574
C03024=1194.008,168.365,-55.720,-178.052,6.338,148.575
C03025=1194.012,168.116,-55.698,-178.055,6.336,148.575
C03026=1194.018,167.867,-55.676,-178.058,6.334,148.575
C03027=1194.023,167.618,-55.654,-178.060,6.333,148.576
C03028=1194.027,167.369,-55.632,-178.063,6.331,148.576
C03029=1194.032,167.120,-55.610,-178.066,6.329,148.576
C03030=1194.036,166.871,-55.588,-178.068,6.328,148.577
C03031=1194.041,166.622,-55.566,-178.071,6.327,148.577
C03032=1194.045,166.373,-55.544,-178.073,6.325,148.578
C03033=1194.050,166.124,-55.523,-178.076,6.323,148.578
C03034=1194.055,165.875,-55.500,-178.079,6.321,148.578
C03035=1194.060,165.626,-55.478,-178.082,6.320,148.579
C03036=1194.064,165.377,-55.456,-178.084,6.318,148.579
C03037=1194.069,165.128,-55.435,-178.087,6.316,148.580
C03038=1194.073,164.879,-55.413,-178.089,6.315,148.580
C03039=1194.078,164.630,-55.391,-178.092,6.313,148.580
C03040=1194.083,164.381,-55.369,-178.094,6.311,148.581
C03041=1194.087,164.132,-55.347,-178.097,6.310,148.581
C03042=1194.092,163.883,-55.325,-178.100,6.308,148.582
C03043=1194.097,163.634,-55.303,-178.103,6.306,148.582
C03044=1194.101,163.385,-55.282,-178.105,6.305,148.582
C03045=1194.106,163.136,-55.260,-178.108,6.304,148.583
C03046=1194.111,162.887,-55.239,-178.110,6.302,148.583
C03047=1194.116,162.638,-55.217,-178.113,6.300,148.584
C03048=1194.120,162.389,-55.195,-178.116,6.298,148.584
C03049=1194.125,162.140,-55.173,-178.118,6.296,148.584
C03050=1194.129,161.891,-55.151,-178.121,6.295,148.585
C03051=1194.134,161.642,-55.130,-178.124,6.294,148.585
C03052=1194.139,161.393,-55.109,-178.126,6.292,148.586
C03053=1194.143,161.144,-55.087,-178.129,6.291,148.586
C03054=1194.148,160.895,-55.065,-178.132,6.289,148.586
C03055=1194.153,160.646,-55.043,-178.134,6.287,148.587
C03056=1194.157,160.397,-55.021,-178.136,6.286,148.587
C03057=1194.163,160.148,-55.000,-178.139,6.284,148.587
C03058=1194.167,159.898,-54.978,-178.142,6.283,148.588
C03059=1194.172,159.650,-54.956,-178.145,6.281,148.588
C03060=1194.177,159.401,-54.935,-178.148,6.279,148.589
C03061=1194.181,159.132,-54.912,-178.150,6.277,148.589
C03062=1194.187,158.863,-54.889,-178.153,6.276,148.590
C03063=1194.192,158.594,-54.866,-178.156,6.274,148.590
C03064=1194.197,158.325,-54.842,-178.159,6.272,148.591
C03065=1194.202,158.076,-54.821,-178.161,6.271,148.591
C03066=1194.206,157.826,-54.799,-178.164,6.269,148.591
C03067=1194.211,157.578,-54.777,-178.166,6.268,148.592
C03068=1194.215,157.329,-54.757,-178.169,6.266,148.592
C03069=1194.220,157.079,-54.735,-178.172,6.265,148.593
C03070=1194.225,156.831,-54.713,-178.175,6.263,148.593
C03071=1194.230,156.581,-54.692,-178.177,6.261,148.593
C03072=1194.235,156.333,-54.670,-178.180,6.260,148.594
C03073=1194.239,156.083,-54.649,-178.182,6.258,148.594
C03074=1194.243,155.835,-54.628,-178.185,6.257,148.595
C03075=1194.248,155.586,-54.606,-178.188,6.255,148.595
C03076=1194.253,155.337,-54.585,-178.191,6.253,148.595
C03077=1194.258,155.087,-54.563,-178.193,6.252,148.596
C03078=1194.263,154.838,-54.542,-178.196,6.251,148.596
C03079=1194.267,154.590,-54.521,-178.198,6.249,148.597
C03080=1194.272,154.340,-54.500,-178.201,6.247,148.597
C03081=1194.276,154.091,-54.478,-178.203,6.246,148.598
C03082=1194.282,153.842,-54.457,-178.206,6.245,148.598
C03083=1194.286,153.593,-54.435,-178.209,6.243,148.598
C03084=1194.291,153.344,-54.415,-178.212,6.241,148.599
C03085=1194.295,153.095,-54.393,-178.214,6.239,148.599
C03086=1194.300,152.846,-54.372,-178.217,6.239,148.600
C03087=1194.306,152.596,-54.351,-178.219,6.237,148.600
C03088=1194.310,152.348,-54.330,-178.222,6.235,148.601
C03089=1194.315,152.099,-54.309,-178.225,6.233,148.601
C03090=1194.319,151.849,-54.287,-178.227,6.232,148.601
C03091=1194.324,151.600,-54.267,-178.230,6.231,148.602
C03092=1194.329,151.351,-54.246,-178.233,6.229,148.602
C03093=1194.334,151.103,-54.224,-178.235,6.227,148.603
C03094=1194.338,150.854,-54.204,-178.238,6.226,148.603
C03095=1194.342,150.604,-54.182,-178.240,6.225,148.603
C03096=1194.347,150.355,-54.161,-178.243,6.223,148.604
C03097=1194.352,150.106,-54.140,-178.246,6.221,148.604
C03098=1194.357,149.857,-54.119,-178.249,6.220,148.605
C03099=1194.362,149.608,-54.098,-178.251,6.219,148.605
C03100=1194.366,149.359,-54.077,-178.254,6.217,148.606
C03101=1194.371,149.109,-54.056,-178.256,6.215,148.606
C03102=1194.376,148.861,-54.034,-178.259,6.214,148.607
C03103=1194.380,148.612,-54.014,-178.262,6.213,148.607
C03104=1194.385,148.362,-53.993,-178.264,6.211,148.607
C03105=1194.390,148.114,-53.972,-178.267,6.209,148.608
C03106=1194.395,147.865,-53.951,-178.270,6.207,148.608
C03107=1194.400,147.616,-53.930,-178.272,6.207,148.609
C03108=1194.404,147.366,-53.909,-178.275,6.205,148.609
C03109=1194.409,147.117,-53.888,-178.278,6.203,148.609
C03110=1194.413,146.868,-53.867,-178.280,6.202,148.610
C03111=1194.418,146.619,-53.846,-178.282,6.201,148.610
C03112=1194.423,146.370,-53.826,-178.286,6.199,148.611
C03113=1194.428,146.121,-53.805,-178.288,6.197,148.611
C03114=1194.433,145.872,-53.784,-178.290,6.196,148.612
C03115=1194.437,145.623,-53.763,-178.293,6.195,148.612
C03116=1194.442,145.374,-53.742,-178.296,6.193,148.613
C03117=1194.447,145.125,-53.721,-178.299,6.191,148.613
C03118=1194.451,144.875,-53.700,-178.301,6.191,148.613
C03119=1194.456,144.626,-53.680,-178.304,6.189,148.614
C03120=1194.461,144.377,-53.659,-178.307,6.187,148.614
C03121=1194.465,144.128,-53.638,-178.309,6.186,148.615
C03122=1194.471,143.879,-53.617,-178.312,6.185,148.615
C03123=1194.475,143.630,-53.597,-178.314,6.183,148.616
C03124=1194.479,143.381,-53.577,-178.317,6.181,148.616
C03125=1194.485,143.132,-53.556,-178.320,6.180,148.617
C03126=1194.489,142.883,-53.535,-178.322,6.179,148.617
C03127=1194.494,142.633,-53.514,-178.325,6.177,148.617
C03128=1194.499,142.384,-53.494,-178.327,6.176,148.618
C03129=1194.504,142.135,-53.473,-178.330,6.175,148.618
C03130=1194.508,141.886,-53.453,-178.333,6.173,148.619
C03131=1194.513,141.637,-53.432,-178.336,6.171,148.619
C03132=1194.518,141.388,-53.411,-178.338,6.170,148.619
C03133=1194.522,141.139,-53.391,-178.341,6.169,148.620
C03134=1194.528,140.890,-53.370,-178.344,6.167,148.620
C03135=1194.532,140.641,-53.350,-178.346,6.166,148.621
C03136=1194.537,140.392,-53.329,-178.348,6.164,148.621
C03137=1194.542,140.143,-53.308,-178.352,6.163,148.622
C03138=1194.546,139.894,-53.288,-178.354,6.162,148.622
C03139=1194.551,139.644,-53.267,-178.356,6.160,148.623
C03140=1194.556,139.395,-53.247,-178.359,6.158,148.623
C03141=1194.560,139.147,-53.226,-178.362,6.158,148.624
C03142=1194.565,138.897,-53.205,-178.364,6.156,148.624
C03143=1194.570,138.648,-53.186,-178.367,6.154,148.624
C03144=1194.574,138.399,-53.165,-178.370,6.152,148.625
C03145=1194.580,138.149,-53.144,-178.372,6.152,148.625
C03146=1194.584,137.901,-53.124,-178.375,6.150,148.626
C03147=1194.588,137.652,-53.103,-178.378,6.148,148.626
C03148=1194.594,137.402,-53.082,-178.380,6.148,148.627
C03149=1194.598,137.153,-53.063,-178.383,6.146,148.627
C03150=1194.603,136.904,-53.042,-178.386,6.144,148.628
C03151=1194.607,136.655,-53.022,-178.388,6.143,148.628
C03152=1194.612,136.406,-53.001,-178.391,6.142,148.629
C03153=1194.617,136.156,-52.981,-178.394,6.140,148.629
C03154=1194.622,135.908,-52.961,-178.396,6.139,148.629
C03155=1194.627,135.659,-52.941,-178.399,6.138,148.630
C03156=1194.632,135.410,-52.920,-178.402,6.136,148.630
C03157=1194.637,135.160,-52.900,-178.404,6.135,148.631
C03158=1194.641,134.911,-52.880,-178.406,6.133,148.631
C03159=1194.645,134.662,-52.860,-178.410,6.132,148.632
C03160=1194.651,134.412,-52.839,-178.412,6.131,148.632
C03161=1194.655,134.163,-52.819,-178.414,6.129,148.633
C03162=1194.660,133.914,-52.799,-178.417,6.128,148.633
C03163=1194.665,133.665,-52.779,-178.420,6.127,148.634
C03164=1194.670,133.416,-52.759,-178.422,6.125,148.634
C03165=1194.675,133.148,-52.737,-178.426,6.123,148.635
C03166=1194.679,132.879,-52.715,-178.428,6.122,148.635
C03167=1194.685,132.610,-52.694,-178.431,6.121,148.636
C03168=1194.690,132.341,-52.671,-178.434,6.119,148.636
C03169=1194.696,132.093,-52.652,-178.436,6.117,148.636
C03170=1194.700,131.844,-52.631,-178.439,6.117,148.637
C03171=1194.705,131.594,-52.612,-178.442,6.115,148.637
C03172=1194.709,131.345,-52.591,-178.444,6.113,148.638
C03173=1194.714,131.096,-52.571,-178.447,6.113,148.638
C03174=1194.718,130.847,-52.551,-178.450,6.111,148.639
C03175=1194.723,130.598,-52.531,-178.452,6.109,148.639
C03176=1194.729,130.349,-52.511,-178.455,6.109,148.640
C03177=1194.733,130.100,-52.491,-178.458,6.107,148.640
C03178=1194.738,129.850,-52.471,-178.460,6.106,148.641
C03179=1194.742,129.601,-52.451,-178.462,6.104,148.641
C03180=1194.748,129.352,-52.431,-178.466,6.103,148.642
C03181=1194.752,129.103,-52.411,-178.468,6.102,148.642
C03182=1194.757,128.854,-52.391,-178.470,6.100,148.642
C03183=1194.762,128.604,-52.372,-178.473,6.099,148.643
C03184=1194.766,128.355,-52.351,-178.476,6.098,148.643
C03185=1194.772,128.106,-52.332,-178.478,6.096,148.644
C03186=1194.776,127.857,-52.312,-178.481,6.095,148.645
C03187=1194.781,127.608,-52.292,-178.484,6.094,148.645
C03188=1194.785,127.359,-52.272,-178.486,6.092,148.645
C03189=1194.790,127.109,-52.252,-178.489,6.091,148.646
C03190=1194.795,126.860,-52.233,-178.492,6.089,148.646
C03191=1194.800,126.611,-52.212,-178.494,6.088,148.647
C03192=1194.804,126.362,-52.193,-178.497,6.087,148.647
C03193=1194.809,126.112,-52.173,-178.500,6.085,148.648
C03194=1194.814,125.864,-52.153,-178.502,6.084,148.648
C03195=1194.819,125.614,-52.133,-178.505,6.083,148.649
C03196=1194.824,125.365,-52.114,-178.507,6.082,148.649
C03197=1194.828,125.116,-52.093,-178.510,6.080,148.650
C03198=1194.833,124.867,-52.074,-178.513,6.079,148.650
C03199=1194.838,124.618,-52.054,-178.515,6.078,148.651
C03200=1194.843,124.369,-52.034,-178.518,6.076,148.651
C03201=1194.848,124.120,-52.015,-178.520,6.076,148.652
C03202=1194.853,123.870,-51.995,-178.523,6.074,148.652
C03203=1194.857,123.621,-51.975,-178.526,6.072,148.653
C03204=1194.863,123.372,-51.955,-178.528,6.071,148.653
C03205=1194.867,123.123,-51.936,-178.531,6.070,148.653
C03206=1194.871,122.874,-51.917,-178.534,6.069,148.654
C03207=1194.876,122.624,-51.897,-178.536,6.067,148.654
C03208=1194.881,122.375,-51.878,-178.538,6.066,148.655
C03209=1194.886,122.126,-51.857,-178.542,6.065,148.655
C03210=1194.891,121.877,-51.838,-178.544,6.063,148.656
C03211=1194.896,121.628,-51.818,-178.546,6.062,148.656
C03212=1194.901,121.378,-51.799,-178.550,6.061,148.657
C03213=1194.905,121.129,-51.780,-178.552,6.060,148.657
C03214=1194.910,120.880,-51.760,-178.555,6.059,148.658
C03215=1194.914,120.631,-51.740,-178.557,6.058,148.658
C03216=1194.919,120.381,-51.720,-178.560,6.056,148.659
C03217=1194.925,120.133,-51.701,-178.563,6.054,148.659
C03218=1194.929,119.883,-51.681,-178.565,6.053,148.660
C03219=1194.934,119.634,-51.663,-178.568,6.052,148.660
C03220=1194.939,119.385,-51.643,-178.570,6.051,148.661
C03221=1194.943,119.135,-51.623,-178.573,6.049,148.661
C03222=1194.949,118.886,-51.604,-178.576,6.049,148.662
C03223=1194.953,118.637,-51.585,-178.578,6.047,148.662
C03224=1194.957,118.388,-51.565,-178.580,6.046,148.663
C03225=1194.963,118.139,-51.546,-178.584,6.045,148.663
C03226=1194.968,117.889,-51.527,-178.586,6.043,148.664
C03227=1194.973,117.640,-51.507,-178.589,6.042,148.664
C03228=1194.977,117.391,-51.488,-178.592,6.041,148.665
C03229=1194.982,117.142,-51.469,-178.594,6.040,148.665
C03230=1194.987,116.893,-51.449,-178.597,6.038,148.666
C03231=1194.992,116.643,-51.430,-178.599,6.037,148.666
C03232=1194.996,116.395,-51.411,-178.602,6.036,148.667
C03233=1195.001,116.145,-51.391,-178.604,6.035,148.667
C03234=1195.006,115.896,-51.372,-178.607,6.033,148.668
C03235=1195.010,115.647,-51.353,-178.610,6.033,148.668
C03236=1195.016,115.398,-51.334,-178.612,6.031,148.669
C03237=1195.020,115.148,-51.314,-178.615,6.030,148.669
C03238=1195.025,114.899,-51.294,-178.618,6.029,148.670
C03239=1195.030,114.650,-51.276,-178.620,6.027,148.670
C03240=1195.035,114.401,-51.256,-178.623,6.026,148.671
C03241=1195.040,114.151,-51.237,-178.626,6.024,148.671
C03242=1195.044,113.902,-51.218,-178.628,6.024,148.672
C03243=1195.050,113.653,-51.199,-178.631,6.022,148.672
C03244=1195.054,113.404,-51.179,-178.633,6.021,148.673
C03245=1195.059,113.155,-51.161,-178.636,6.020,148.673
C03246=1195.064,112.905,-51.141,-178.638,6.019,148.674
C03247=1195.069,112.656,-51.123,-178.642,6.017,148.674
C03248=1195.073,112.407,-51.103,-178.644,6.017,148.675
C03249=1195.079,112.158,-51.084,-178.646,6.015,148.675
C03250=1195.083,111.909,-51.065,-178.649,6.014,148.676
C03251=1195.088,111.660,-51.046,-178.652,6.012,148.676
C03252=1195.092,111.410,-51.027,-178.654,6.012,148.677
C03253=1195.098,111.161,-51.008,-178.657,6.010,148.677
C03254=1195.102,110.911,-50.988,-178.659,6.009,148.678
C03255=1195.107,110.663,-50.970,-178.662,6.008,148.678
C03256=1195.112,110.413,-50.951,-178.665,6.007,148.679
C03257=1195.117,110.164,-50.932,-178.668,6.005,148.679
C03258=1195.121,109.914,-50.912,-178.670,6.005,148.680
C03259=1195.126,109.665,-50.894,-178.673,6.003,148.680
C03260=1195.132,109.416,-50.875,-178.675,6.002,148.681
C03261=1195.136,109.167,-50.856,-178.678,6.000,148.681
C03262=1195.141,108.918,-50.838,-178.680,6.000,148.682
C03263=1195.145,108.668,-50.818,-178.683,5.998,148.682
C03264=1195.151,108.420,-50.799,-178.686,5.998,148.683
C03265=1195.155,108.170,-50.781,-178.689,5.996,148.683
C03266=1195.160,107.921,-50.762,-178.691,5.995,148.684
C03267=1195.164,107.672,-50.742,-178.694,5.993,148.684
C03268=1195.170,107.422,-50.724,-178.696,5.993,148.685
C03269=1195.175,107.154,-50.704,-178.699,5.991,148.685
C03270=1195.180,106.885,-50.683,-178.702,5.991,148.686
C03271=1195.185,106.617,-50.663,-178.704,5.989,148.686
C03272=1195.191,106.349,-50.643,-178.708,5.987,148.687
C03273=1195.195,106.099,-50.624,-178.710,5.987,148.688
C03274=1195.200,105.850,-50.606,-178.713,5.985,148.688
C03275=1195.205,105.601,-50.586,-178.715,5.984,148.688
C03276=1195.210,105.351,-50.568,-178.718,5.983,148.689
C03277=1195.215,105.103,-50.549,-178.720,5.982,148.689
C03278=1195.220,104.853,-50.530,-178.724,5.980,148.690
C03279=1195.224,104.604,-50.512,-178.726,5.980,148.691
C03280=1195.230,104.355,-50.493,-178.729,5.978,148.691
C03281=1195.234,104.105,-50.474,-178.731,5.977,148.692
C03282=1195.239,103.856,-50.455,-178.734,5.977,148.692
C03283=1195.243,103.607,-50.436,-178.736,5.975,148.693
C03284=1195.248,103.358,-50.418,-178.739,5.974,148.693
C03285=1195.254,103.109,-50.399,-178.742,5.973,148.694
C03286=1195.258,102.859,-50.381,-178.744,5.972,148.694
C03287=1195.263,102.610,-50.362,-178.747,5.970,148.695
C03288=1195.268,102.361,-50.343,-178.749,5.969,148.695
C03289=1195.273,102.111,-50.325,-178.752,5.968,148.696
C03290=1195.277,101.862,-50.306,-178.754,5.967,148.696
C03291=1195.283,101.613,-50.288,-178.758,5.966,148.697
C03292=1195.287,101.363,-50.270,-178.760,5.965,148.697
C03293=1195.292,101.114,-50.251,-178.762,5.964,148.698
C03294=1195.297,100.865,-50.232,-178.765,5.962,148.698
C03295=1195.302,100.616,-50.214,-178.768,5.962,148.699
C03296=1195.306,100.366,-50.195,-178.770,5.960,148.699
C03297=1195.311,100.117,-50.177,-178.773,5.960,148.700
C03298=1195.317,99.868,-50.158,-178.776,5.958,148.700
C03299=1195.321,99.619,-50.140,-178.778,5.957,148.701
C03300=1195.326,99.369,-50.122,-178.781,5.956,148.701
C03301=1195.331,99.120,-50.103,-178.784,5.955,148.702
C03302=1195.336,98.871,-50.084,-178.786,5.954,148.703
C03303=1195.340,98.621,-50.066,-178.789,5.953,148.703
C03304=1195.345,98.372,-50.048,-178.791,5.952,148.704
C03305=1195.351,98.123,-50.029,-178.794,5.950,148.704
C03306=1195.355,97.874,-50.010,-178.796,5.949,148.705
C03307=1195.360,97.624,-49.992,-178.799,5.949,148.705
C03308=1195.365,97.375,-49.974,-178.802,5.947,148.706
C03309=1195.370,97.126,-49.956,-178.804,5.946,148.706
C03310=1195.375,96.877,-49.937,-178.807,5.945,148.707
C03311=1195.379,96.627,-49.919,-178.810,5.944,148.707
C03312=1195.384,96.378,-49.901,-178.812,5.942,148.708
C03313=1195.389,96.129,-49.883,-178.815,5.942,148.708
C03314=1195.394,95.880,-49.865,-178.817,5.941,148.709
C03315=1195.398,95.630,-49.847,-178.820,5.940,148.710
C03316=1195.404,95.381,-49.827,-178.823,5.939,148.710
C03317=1195.409,95.132,-49.809,-178.826,5.937,148.711
C03318=1195.414,94.883,-49.791,-178.828,5.936,148.711
C03319=1195.418,94.633,-49.773,-178.831,5.936,148.712
C03320=1195.423,94.384,-49.755,-178.833,5.934,148.712
C03321=1195.428,94.134,-49.737,-178.836,5.933,148.713
C03322=1195.433,93.885,-49.719,-178.839,5.932,148.713
C03323=1195.438,93.636,-49.700,-178.841,5.931,148.714
C03324=1195.443,93.387,-49.682,-178.843,5.930,148.714
C03325=1195.447,93.137,-49.664,-178.846,5.929,148.715
C03326=1195.452,92.888,-49.646,-178.849,5.928,148.715
C03327=1195.457,92.639,-49.627,-178.852,5.927,148.716
C03328=1195.462,92.390,-49.609,-178.854,5.926,148.716
C03329=1195.467,92.141,-49.591,-178.857,5.925,148.717
C03330=1195.472,91.891,-49.573,-178.859,5.923,148.717
C03331=1195.476,91.642,-49.555,-178.862,5.923,148.718
C03332=1195.481,91.392,-49.537,-178.864,5.922,148.718
C03333=1195.486,91.143,-49.519,-178.867,5.920,148.719
C03334=1195.491,90.894,-49.501,-178.869,5.919,148.720
C03335=1195.496,90.644,-49.484,-178.873,5.918,148.720
C03336=1195.501,90.395,-49.466,-178.875,5.917,148.721
C03337=1195.506,90.146,-49.448,-178.877,5.917,148.721
C03338=1195.511,89.897,-49.430,-178.881,5.915,148.722
C03339=1195.515,89.647,-49.412,-178.883,5.914,148.722
C03340=1195.520,89.398,-49.394,-178.886,5.913,148.723
C03341=1195.525,89.148,-49.376,-178.888,5.912,148.723
C03342=1195.530,88.899,-49.358,-178.891,5.911,148.724
C03343=1195.535,88.650,-49.340,-178.893,5.910,148.724
C03344=1195.540,88.401,-49.322,-178.896,5.909,148.725
C03345=1195.545,88.152,-49.304,-178.898,5.908,148.726
C03346=1195.550,87.902,-49.287,-178.901,5.907,148.726
C03347=1195.555,87.653,-49.269,-178.903,5.906,148.727
C03348=1195.560,87.404,-49.251,-178.906,5.905,148.727
C03349=1195.564,87.154,-49.232,-178.909,5.904,148.728
C03350=1195.569,86.905,-49.214,-178.911,5.903,148.728
C03351=1195.574,86.655,-49.196,-178.914,5.903,148.729
C03352=1195.579,86.406,-49.179,-178.917,5.901,148.729
C03353=1195.584,86.156,-49.161,-178.919,5.900,148.730
C03354=1195.589,85.907,-49.143,-178.922,5.899,148.730
C03355=1195.594,85.658,-49.125,-178.925,5.898,148.731
C03356=1195.599,85.409,-49.107,-178.927,5.897,148.732
C03357=1195.603,85.159,-49.090,-178.930,5.896,148.732
C03358=1195.608,84.910,-49.072,-178.932,5.895,148.733
C03359=1195.613,84.661,-49.054,-178.935,5.894,148.733
C03360=1195.618,84.412,-49.036,-178.937,5.892,148.734
C03361=1195.623,84.162,-49.019,-178.940,5.892,148.734
C03362=1195.628,83.913,-49.001,-178.943,5.891,148.735
C03363=1195.633,83.664,-48.983,-178.945,5.890,148.735
C03364=1195.637,83.414,-48.967,-178.948,5.889,148.736
C03365=1195.642,83.165,-48.949,-178.950,5.888,148.736
C03366=1195.647,82.916,-48.931,-178.953,5.887,148.737
C03367=1195.652,82.666,-48.913,-178.956,5.886,148.738
C03368=1195.657,82.417,-48.895,-178.958,5.885,148.738
C03369=1195.662,82.168,-48.877,-178.961,5.884,148.739
C03370=1195.667,81.918,-48.861,-178.964,5.883,148.739
C03371=1195.672,81.669,-48.843,-178.966,5.882,148.740
C03372=1195.676,81.420,-48.825,-178.969,5.881,148.740
C03373=1195.682,81.151,-48.806,-178.971,5.880,148.741
C03374=1195.687,80.883,-48.787,-178.975,5.879,148.742
C03375=1195.693,80.615,-48.768,-178.977,5.878,148.742
C03376=1195.698,80.346,-48.750,-178.980,5.877,148.743
C03377=1195.702,80.097,-48.732,-178.983,5.876,148.743
C03378=1195.707,79.848,-48.714,-178.985,5.875,148.744
C03379=1195.713,79.598,-48.697,-178.988,5.874,148.744
C03380=1195.718,79.349,-48.679,-178.991,5.873,148.745
C03381=1195.722,79.099,-48.662,-178.993,5.872,148.746
C03382=1195.727,78.850,-48.644,-178.995,5.872,148.746
C03383=1195.732,78.600,-48.627,-178.998,5.870,148.747
C03384=1195.736,78.351,-48.610,-179.001,5.869,148.747
C03385=1195.742,78.102,-48.592,-179.003,5.869,148.748
C03386=1195.746,77.852,-48.574,-179.006,5.867,148.748
C03387=1195.752,77.603,-48.557,-179.009,5.867,148.749
C03388=1195.756,77.355,-48.540,-179.011,5.866,148.749
C03389=1195.762,77.105,-48.523,-179.014,5.864,148.750
C03390=1195.767,76.856,-48.505,-179.016,5.863,148.751
C03391=1195.771,76.606,-48.488,-179.019,5.863,148.751
C03392=1195.776,76.356,-48.471,-179.021,5.862,148.752
C03393=1195.781,76.107,-48.453,-179.024,5.861,148.752
C03394=1195.786,75.858,-48.436,-179.027,5.860,148.753
C03395=1195.791,75.608,-48.418,-179.029,5.859,148.753
C03396=1195.795,75.359,-48.402,-179.032,5.858,148.754
C03397=1195.801,75.110,-48.385,-179.035,5.857,148.755
C03398=1195.806,74.861,-48.367,-179.037,5.856,148.755
C03399=1195.810,74.611,-48.350,-179.040,5.856,148.756
C03400=1195.815,74.362,-48.332,-179.042,5.854,148.756
C03401=1195.820,74.112,-48.315,-179.045,5.853,148.757
C03402=1195.825,73.863,-48.298,-179.047,5.853,148.757
C03403=1195.830,73.614,-48.280,-179.050,5.851,148.758
C03404=1195.835,73.365,-48.264,-179.053,5.851,148.759
C03405=1195.840,73.115,-48.247,-179.055,5.850,148.759
C03406=1195.845,72.865,-48.229,-179.058,5.849,148.760
C03407=1195.849,72.616,-48.212,-179.061,5.848,148.760
C03408=1195.855,72.367,-48.195,-179.063,5.847,148.761
C03409=1195.859,72.117,-48.178,-179.066,5.846,148.761
C03410=1195.865,71.869,-48.161,-179.069,5.845,148.762
C03411=1195.869,71.619,-48.144,-179.071,5.844,148.762
C03412=1195.874,71.369,-48.127,-179.074,5.843,148.763
C03413=1195.879,71.120,-48.110,-179.076,5.843,148.764
C03414=1195.884,70.871,-48.092,-179.079,5.841,148.764
C03415=1195.889,70.622,-48.076,-179.082,5.841,148.765
C03416=1195.894,70.372,-48.058,-179.084,5.840,148.765
C03417=1195.899,70.123,-48.042,-179.086,5.839,148.766
C03418=1195.904,69.873,-48.024,-179.089,5.837,148.766
C03419=1195.908,69.624,-48.007,-179.092,5.837,148.767
C03420=1195.914,69.375,-47.990,-179.094,5.836,148.768
C03421=1195.918,69.125,-47.973,-179.096,5.835,148.768
C03422=1195.923,68.876,-47.956,-179.100,5.834,148.769
C03423=1195.928,68.626,-47.940,-179.102,5.834,148.769
C03424=1195.934,68.377,-47.923,-179.104,5.833,148.770
C03425=1195.938,68.127,-47.906,-179.107,5.832,148.771
C03426=1195.943,67.878,-47.888,-179.110,5.830,148.771
C03427=1195.948,67.629,-47.871,-179.112,5.830,148.772
C03428=1195.952,67.379,-47.855,-179.115,5.829,148.772
C03429=1195.958,67.130,-47.838,-179.117,5.828,148.773
C03430=1195.962,66.881,-47.821,-179.120,5.827,148.773
C03431=1195.968,66.631,-47.804,-179.123,5.827,148.774
C03432=1195.973,66.382,-47.788,-179.125,5.826,148.775
C03433=1195.978,66.132,-47.770,-179.128,5.825,148.775
C03434=1195.982,65.883,-47.754,-179.130,5.824,148.776
C03435=1195.987,65.633,-47.737,-179.133,5.823,148.776
C03436=1195.993,65.384,-47.720,-179.136,5.822,148.777
C03437=1195.997,65.135,-47.703,-179.138,5.821,148.777
C03438=1196.002,64.885,-47.687,-179.141,5.821,148.778
C03439=1196.007,64.636,-47.670,-179.144,5.819,148.779
C03440=1196.012,64.387,-47.653,-179.146,5.819,148.779
C03441=1196.017,64.137,-47.636,-179.149,5.818,148.780
C03442=1196.022,63.887,-47.619,-179.151,5.817,148.780
C03443=1196.027,63.639,-47.603,-179.154,5.816,148.781
C03444=1196.032,63.389,-47.586,-179.157,5.815,148.782
C03445=1196.036,63.139,-47.569,-179.159,5.815,148.782
C03446=1196.042,62.891,-47.553,-179.161,5.814,148.783
C03447=1196.047,62.641,-47.535,-179.164,5.813,148.783
C03448=1196.051,62.391,-47.519,-179.167,5.812,148.784
C03449=1196.056,62.143,-47.502,-179.169,5.811,148.784
C03450=1196.061,61.893,-47.486,-179.172,5.810,148.785
C03451=1196.066,61.643,-47.468,-179.174,5.810,148.785
C03452=1196.071,61.395,-47.452,-179.177,5.809,148.786
C03453=1196.076,61.144,-47.436,-179.180,5.808,148.787
C03454=1196.081,60.895,-47.419,-179.182,5.807,148.787
C03455=1196.086,60.646,-47.403,-179.185,5.806,148.788
C03456=1196.091,60.396,-47.386,-179.187,5.806,148.789
C03457=1196.096,60.148,-47.370,-179.189,5.805,148.789
C03458=1196.101,59.898,-47.352,-179.193,5.803,148.790
C03459=1196.106,59.648,-47.336,-179.195,5.803,148.790
C03460=1196.111,59.399,-47.320,-179.197,5.802,148.791
C03461=1196.115,59.149,-47.303,-179.200,5.801,148.791
C03462=1196.121,58.900,-47.287,-179.203,5.801,148.792
C03463=1196.126,58.651,-47.270,-179.205,5.799,148.793
C03464=1196.130,58.401,-47.254,-179.208,5.799,148.793
C03465=1196.135,58.152,-47.238,-179.211,5.798,148.794
C03466=1196.140,57.902,-47.221,-179.213,5.797,148.794
C03467=1196.146,57.653,-47.204,-179.216,5.797,148.795
C03468=1196.151,57.403,-47.188,-179.219,5.795,148.796
C03469=1196.155,57.154,-47.171,-179.221,5.794,148.796
C03470=1196.160,56.905,-47.155,-179.224,5.794,148.797
C03471=1196.165,56.656,-47.138,-179.226,5.793,148.797
C03472=1196.170,56.406,-47.123,-179.228,5.792,148.798
C03473=1196.175,56.156,-47.106,-179.231,5.792,148.799
C03474=1196.180,55.908,-47.089,-179.234,5.791,148.799
C03475=1196.185,55.657,-47.073,-179.236,5.790,148.800
C03476=1196.190,55.408,-47.057,-179.239,5.789,148.800
C03477=1196.195,55.139,-47.040,-179.242,5.789,148.801
C03478=1196.200,54.872,-47.022,-179.245,5.787,148.802
C03479=1196.206,54.602,-47.004,-179.247,5.787,148.802
C03480=1196.211,54.334,-46.986,-179.250,5.786,148.803
C03481=1196.217,54.085,-46.971,-179.253,5.784,148.803
C03482=1196.221,53.835,-46.954,-179.255,5.784,148.804
C03483=1196.226,53.587,-46.938,-179.258,5.783,148.805
C03484=1196.231,53.336,-46.922,-179.260,5.783,148.805
C03485=1196.236,53.088,-46.905,-179.263,5.782,148.806
C03486=1196.241,52.838,-46.889,-179.265,5.781,148.806
C03487=1196.245,52.588,-46.873,-179.268,5.780,148.807
C03488=1196.250,52.339,-46.856,-179.271,5.779,148.808
C03489=1196.255,52.089,-46.841,-179.273,5.779,148.808
C03490=1196.260,51.840,-46.824,-179.276,5.778,148.809
C03491=1196.265,51.590,-46.808,-179.278,5.777,148.809
C03492=1196.271,51.341,-46.791,-179.281,5.777,148.810
C03493=1196.276,51.092,-46.776,-179.283,5.776,148.810
C03494=1196.281,50.842,-46.759,-179.286,5.774,148.811
C03495=1196.286,50.593,-46.744,-179.289,5.774,148.812
C03496=1196.291,50.343,-46.727,-179.291,5.773,148.812
C03497=1196.296,50.094,-46.711,-179.294,5.773,148.813
C03498=1196.301,49.845,-46.695,-179.296,5.772,148.814
C03499=1196.306,49.595,-46.679,-179.299,5.771,148.814
C03500=1196.310,49.346,-46.662,-179.301,5.771,148.815
C03501=1196.316,49.096,-46.647,-179.304,5.769,148.815
C03502=1196.320,48.846,-46.631,-179.307,5.769,148.816
C03503=1196.325,48.598,-46.615,-179.309,5.768,148.816
C03504=1196.330,48.348,-46.599,-179.312,5.767,148.817
C03505=1196.335,48.099,-46.583,-179.314,5.767,148.818
C03506=1196.340,47.849,-46.567,-179.317,5.766,148.818
C03507=1196.345,47.600,-46.551,-179.319,5.765,148.819
C03508=1196.350,47.351,-46.535,-179.322,5.764,148.820
C03509=1196.355,47.100,-46.519,-179.325,5.763,148.820
C03510=1196.360,46.852,-46.503,-179.327,5.763,148.821
C03511=1196.365,46.602,-46.487,-179.330,5.762,148.821
C03512=1196.370,46.352,-46.471,-179.332,5.762,148.822
C03513=1196.375,46.103,-46.455,-179.335,5.761,148.822
C03514=1196.380,45.853,-46.439,-179.337,5.760,148.823
C03515=1196.385,45.604,-46.423,-179.340,5.760,148.824
C03516=1196.390,45.355,-46.408,-179.343,5.758,148.824
C03517=1196.394,45.105,-46.392,-179.345,5.757,148.825
C03518=1196.400,44.856,-46.376,-179.348,5.757,148.826
C03519=1196.404,44.606,-46.359,-179.351,5.756,148.826
C03520=1196.410,44.357,-46.344,-179.353,5.755,148.827
C03521=1196.415,44.108,-46.328,-179.355,5.755,148.827
C03522=1196.420,43.857,-46.312,-179.358,5.754,148.828
C03523=1196.424,43.609,-46.297,-179.360,5.753,148.829
C03524=1196.430,43.360,-46.281,-179.363,5.753,148.829
C03525=1196.434,43.110,-46.265,-179.366,5.752,148.830
C03526=1196.440,42.860,-46.249,-179.369,5.751,148.831
C03527=1196.445,42.611,-46.233,-179.371,5.750,148.831
C03528=1196.450,42.361,-46.217,-179.373,5.750,148.832
C03529=1196.454,42.112,-46.202,-179.376,5.749,148.832
C03530=1196.460,41.863,-46.187,-179.378,5.748,148.833
C03531=1196.464,41.613,-46.171,-179.381,5.748,148.833
C03532=1196.470,41.364,-46.154,-179.383,5.747,148.834
C03533=1196.475,41.114,-46.139,-179.386,5.747,148.835
C03534=1196.479,40.865,-46.123,-179.388,5.746,148.835
C03535=1196.484,40.615,-46.108,-179.392,5.744,148.836
C03536=1196.490,40.366,-46.092,-179.394,5.744,148.837
C03537=1196.495,40.116,-46.076,-179.396,5.743,148.837
C03538=1196.499,39.867,-46.061,-179.399,5.743,148.838
C03539=1196.504,39.618,-46.045,-179.402,5.742,148.838
C03540=1196.509,39.368,-46.029,-179.404,5.741,148.839
C03541=1196.514,39.118,-46.013,-179.406,5.741,148.839
C03542=1196.519,38.869,-45.998,-179.409,5.740,148.840
C03543=1196.524,38.620,-45.983,-179.412,5.740,148.841
C03544=1196.529,38.370,-45.967,-179.414,5.739,148.841
C03545=1196.535,38.120,-45.951,-179.416,5.738,148.842
C03546=1196.539,37.871,-45.936,-179.419,5.738,148.843
C03547=1196.545,37.622,-45.921,-179.422,5.736,148.843
C03548=1196.549,37.372,-45.905,-179.424,5.735,148.844
C03549=1196.554,37.123,-45.890,-179.427,5.735,148.844
C03550=1196.560,36.873,-45.874,-179.430,5.734,148.845
C03551=1196.565,36.624,-45.859,-179.432,5.734,148.846
C03552=1196.569,36.374,-45.843,-179.435,5.733,148.846
C03553=1196.574,36.125,-45.828,-179.437,5.732,148.847
C03554=1196.580,35.875,-45.812,-179.440,5.732,148.848
C03555=1196.584,35.626,-45.797,-179.442,5.731,148.848
C03556=1196.589,35.376,-45.781,-179.445,5.731,148.849
C03557=1196.595,35.127,-45.766,-179.447,5.730,148.849
C03558=1196.599,34.878,-45.751,-179.450,5.730,148.850
C03559=1196.605,34.628,-45.735,-179.452,5.729,148.850
C03560=1196.609,34.378,-45.719,-179.455,5.728,148.851
C03561=1196.614,34.129,-45.704,-179.458,5.727,148.852
C03562=1196.619,33.880,-45.688,-179.461,5.726,148.853
C03563=1196.624,33.630,-45.673,-179.463,5.725,148.853
C03564=1196.629,33.381,-45.658,-179.465,5.725,148.854
C03565=1196.635,33.130,-45.643,-179.468,5.724,148.854
C03566=1196.639,32.881,-45.628,-179.471,5.724,148.855
C03567=1196.645,32.632,-45.612,-179.473,5.723,148.855
C03568=1196.649,32.383,-45.597,-179.475,5.722,148.856
C03569=1196.655,32.133,-45.581,-179.478,5.722,148.857
C03570=1196.659,31.884,-45.566,-179.481,5.721,148.857
C03571=1196.664,31.634,-45.551,-179.483,5.721,148.858
C03572=1196.670,31.384,-45.536,-179.486,5.720,148.859
C03573=1196.674,31.135,-45.521,-179.488,5.719,148.859
C03574=1196.680,30.886,-45.505,-179.491,5.719,148.860
C03575=1196.684,30.637,-45.490,-179.493,5.718,148.860
C03576=1196.690,30.387,-45.475,-179.496,5.718,148.861
C03577=1196.694,30.137,-45.459,-179.498,5.717,148.862
C03578=1196.700,29.887,-45.444,-179.501,5.717,148.862
C03579=1196.704,29.638,-45.429,-179.503,5.716,148.863
C03580=1196.710,29.389,-45.414,-179.506,5.715,148.864
C03581=1196.715,29.120,-45.398,-179.509,5.714,148.864
C03582=1196.720,28.852,-45.381,-179.512,5.713,148.865
C03583=1196.725,28.583,-45.365,-179.514,5.713,148.866
C03584=1196.731,28.314,-45.349,-179.517,5.712,148.866
C03585=1196.736,28.065,-45.334,-179.520,5.712,148.867
C03586=1196.741,27.815,-45.318,-179.522,5.711,148.868
C03587=1196.746,27.566,-45.304,-179.524,5.710,148.868
C03588=1196.751,27.315,-45.288,-179.527,5.710,148.869
C03589=1196.756,27.066,-45.273,-179.530,5.709,148.869
C03590=1196.761,26.816,-45.258,-179.532,5.709,148.870
C03591=1196.766,26.567,-45.243,-179.534,5.708,148.871
C03592=1196.771,26.318,-45.228,-179.537,5.707,148.871
C03593=1196.776,26.068,-45.213,-179.540,5.707,148.872
C03594=1196.781,25.819,-45.198,-179.542,5.706,148.873
C03595=1196.786,25.570,-45.183,-179.545,5.706,148.873
C03596=1196.791,25.320,-45.169,-179.547,5.705,148.874
C03597=1196.797,25.070,-45.153,-179.550,5.705,148.874
C03598=1196.801,24.821,-45.138,-179.552,5.704,148.875
C03599=1196.806,24.572,-45.124,-179.555,5.703,148.876
C03600=1196.811,24.322,-45.108,-179.557,5.703,148.876
C03601=1196.816,24.072,-45.093,-179.560,5.702,148.877
C03602=1196.821,23.822,-45.078,-179.563,5.702,148.878
C03603=1196.826,23.573,-45.063,-179.565,5.701,148.878
C03604=1196.831,23.324,-45.049,-179.567,5.700,148.879
C03605=1196.836,23.074,-45.033,-179.570,5.700,148.879
C03606=1196.841,22.825,-45.019,-179.573,5.699,148.880
C03607=1196.846,22.575,-45.004,-179.575,5.699,148.881
C03608=1196.852,22.325,-44.989,-179.577,5.698,148.881
C03609=1196.856,22.076,-44.974,-179.580,5.697,148.882
C03610=1196.861,21.827,-44.960,-179.583,5.697,148.883
C03611=1196.867,21.577,-44.944,-179.585,5.696,148.883
C03612=1196.872,21.328,-44.930,-179.588,5.695,148.884
C03613=1196.876,21.078,-44.915,-179.590,5.695,148.884
C03614=1196.882,20.828,-44.900,-179.593,5.694,148.885
C03615=1196.887,20.579,-44.885,-179.596,5.694,148.886
C03616=1196.892,20.330,-44.871,-179.598,5.693,148.886
C03617=1196.896,20.081,-44.856,-179.600,5.693,148.887
C03618=1196.902,19.830,-44.841,-179.603,5.692,148.888
C03619=1196.907,19.581,-44.826,-179.606,5.692,148.888
C03620=1196.912,19.332,-44.811,-179.608,5.691,148.889
C03621=1196.917,19.082,-44.797,-179.610,5.690,148.889
C03622=1196.922,18.833,-44.782,-179.613,5.690,148.890
C03623=1196.927,18.583,-44.767,-179.616,5.689,148.891
C03624=1196.932,18.334,-44.752,-179.618,5.689,148.891
C03625=1196.936,18.084,-44.738,-179.621,5.688,148.892
C03626=1196.942,17.834,-44.723,-179.623,5.687,148.893
C03627=1196.947,17.585,-44.708,-179.626,5.687,148.893
C03628=1196.952,17.335,-44.694,-179.628,5.686,148.894
C03629=1196.957,17.086,-44.680,-179.631,5.686,148.895
C03630=1196.963,16.837,-44.664,-179.633,5.685,148.895
C03631=1196.968,16.587,-44.650,-179.636,5.684,148.896
C03632=1196.973,16.337,-44.636,-179.639,5.684,148.896
C03633=1196.977,16.088,-44.621,-179.641,5.683,148.897
C03634=1196.982,15.839,-44.607,-179.643,5.683,148.898
C03635=1196.987,15.589,-44.592,-179.646,5.682,148.898
C03636=1196.993,15.339,-44.577,-179.649,5.682,148.899
C03637=1196.998,15.090,-44.562,-179.651,5.681,148.900
C03638=1197.002,14.840,-44.548,-179.654,5.681,148.900
C03639=1197.007,14.590,-44.534,-179.656,5.680,148.901
C03640=1197.012,14.341,-44.519,-179.659,5.679,148.901
C03641=1197.017,14.092,-44.505,-179.661,5.679,148.902
C03642=1197.023,13.842,-44.490,-179.664,5.678,148.903
C03643=1197.028,13.593,-44.476,-179.666,5.677,148.903
C03644=1197.033,13.343,-44.461,-179.669,5.677,148.904
C03645=1197.038,13.094,-44.447,-179.672,5.676,148.905
C03646=1197.043,12.844,-44.432,-179.674,5.676,148.905
C03647=1197.048,12.594,-44.418,-179.676,5.676,148.906
